(* CODESYS project silver-waffle
   Author: Robert Budgen
   Company: Burkert
   DefaultNamespace: Burkert
   LanguageModelAttribute: qualified-access-only
   Placeholder: Burkert
   Title: Burkert Device Library
   Version: 1.0.0.42

Project tree, tasks and I/O mapping:
  libraries: CAA Types Extern, 3.5.17.0 (CAA Technical Workgroup); CAA Behaviour Model, 3.5.19.0 (CAA Technical Workgroup); CAA FB Factory, 3.5.19.0 (CAA Technical Workgroup); Standard, 3.5.18.0 (System); Util, 3.5.21.0 (System); CmpBitmapPool, 3.5.17.0 (System); VisuDialogs, * (System); MemoryUtils, 3.5.18.0 (3S - Smart Software Solutions GmbH); CAA Memory, 3.5.17.0 (CAA Technical Workgroup); SysTimeRtc, 3.5.20.0 (System); CAA CiA 405, 4.1.0.0 (CAA Technical Workgroup); IoDrvEtherNetIPAdapter, 4.7.0.0 (CODESYS); IoDrvEtherNetIP, 4.7.0.0 (CODESYS); BUILDING, 1.0.0.0 (OSCAT); BASIC, 3.3.4.0 (OSCAT); FloatingPointUtils, 3.5.21.0 (System); 3S CANopenStack, 4.3.0.0 (CODESYS); IoDrvModbusTCP, 4.4.0.0 (CODESYS); Recipe Management, * (System)
  00000000-0000-0000-0000-000000000000|D:\CoDeSys\LibrariesV3\trunk\Intern\CAA\CAA Template\3.2.0.3 draft\Prefix.pdf
  00000000-0000-0000-0000-000000000000|D:\CoDeSys\LibrariesV3\trunk\Intern\CAA\CAA Template\3.4.0.0 draft\Placeholder.xml
  00000000-0000-0000-0000-000000000000|D:\CoDeSys\LibrariesV3\trunk\Intern\CAA\CAA Template\3.5.2.0 draft\Placeholder.xml
  10 Documentation/
    AL1342
    ASi_8694
    Burkert_8050
    CanOpen_8694
  20 Program Organization Units/
    function block ACV_Temp_Loop_UDFB [CFC]
    function block Basic_Temp_LOOP [CFC]
    function block BCV_Temp_Loop_UDFB [CFC]
    function block FIT_DINT_UDBF [LD]
    function block FLOWave_UDFB [CFC]: Alarms, Translate
    Helpers/
      function block CalculateFrequencyWithTime [ST]
      function block Count_to_Hz [CFC]
      function block FB_DilutionCalculator [ST]
      function block FB_LookUp_Table [ST]: GetVarY
      function block FB_TempCorrection [ST]: GetCorrection
      function Flow_ETA [ST]
      program PLC_TIME [ST]
      function RCP_Manager [ST]: LoadAndWrite, ReadAndSave
      function block Virtual_FIT [CFC]
    HMI_Sync/
      Level_0/
        CanOpen/
        eDip/
        function HMI_8228_Sync [ST]
        function block HMI_8605_Sync [ST]
        function HMI_8653_Sync [ST]
        function HMI_ME44AI_Sync [ST]
        function HMI_ME64_Sync [ST]
      Level_1/
        function block ACV_HMI_Sync_UDFB [?]
        function block AIT_HMI_Sync_UDFB [?]
        ASi/
        function block B8050_HMI_Sync_UDFB [?]
        function block BCV_HMI_Sync_UDFB [?]
        function block c8691_HMI_Sync_UDFB [?]
        function block c8694_HMI_Sync_UDFB [?]
        CanOpen/
        function block Contactor_HMI_Sync_UDFB [?]
        function block DI_HMI_Sync_UDFB [?]
        function block DO_HMI_Sync_UDFB [?]
        eDip/
        function block eDip_s8228_HMI_Sync [?]
        function block FB_HMIAlarmBinder [ST]
        function block FIT_HMI_Sync_UDFB [?]
        function block s336x_HMI_Sync [?]
        function block s8050_HMI_Sync [?]
        function block s8098_HMI_Sync_UDFB [?]
        function block s8312_HMI_Sync [?]
        function block s8412_HMI_Sync [?]
        function block SV_HMI_Sync [?]
        VFDs/
      Level_2/
        function block Chase_HMI_Sync_UDFB [?]
        function block Condensate_HMI_Sync_UDFB [?]
        function block PID_HMI_Sync_UDFB [?]
        function block Quick_Mix_HMI_Sync_UDFB [?]
        function block SW_HMI_Sync_UDFB [?]
      Level_3/
        function block Brite_HMI_Sync [?]
        function block Fermenter_HMI_Sync [?]
    Level_0_Remote_IO/
      Advantech/
        function Adam_6015_FB [LD]
        function Adam_6050_FB [LD]
        function Adam_6217_FB [LD]
        function Adam_6250 [ST]
        function Adam_6266_FB [LD]
      ASI/
        function block AC2916_AIT [LD]
      Burkert/
        function eDip_8653_UDFB [?]
        function block eDip_ME64_CTRL [ST]
        function block eDip_ReadDDO [ST]
        function block eDip_ReadDSO [ST]
        function block eDip_ReadSingleItem [ST]
        function block eDip_WriteSingleItem [ST]
        function block ME43_SDO [ST]
        function ME44_DI [ST]
      CanOpen/
        function block CanOpen_8605 [ST]
        function block CanOpen_8653 [ST]
        function block CanOpen_ME64 [ST]
        data type cSDO_DUT
      eDip/
        function block eDip_8605_CTRL [ST]
        function eDip_ME44_AI [ST]
        function eDip_ME44_AO [ST]
        function eDip_ME44_DI [ST]
        function eDip_ME44_DO_Analog [ST]
        function eDip_ME44_DO [ST]
        function block Parse_DDO [ST]
        function block Parse_DSO [ST]
      IFM/
        function block AL1340_UDFB [ST]
        function block AL1342_UDFB [ST]
      Stride/
        function block MB0_RTD [ST]
        function block SIO_MB12CDR [ST]
      Wago/
        function Wago_750_1405 [ST]
        function Wago_750_1504 [ST]
        function Wago_750_496 [ST]
        function Wago_750_555 [ST]
    Level_1_Devices/
      Asi/
        function block ACV_ASI_CTRL_UDFB [?]
        function block B8681_ASI_UDFB [CFC]
        function block BCV_ASI_CTRL_UDFB [?]
      Base_Functions/
        function block Analog_Alarm_UDFB [ST]
        function block Analog_Sensor_UDFB [?]
        function block Basic_ACV_UDFB [?]
        function block Basic_BCV_UDFB [ST]
        function block Basic_FIT [?]
        function block BCV_CTRL_UDFB [?]
        function block Contactor_Control_UDFB [CFC]
        function block DI_UDFB [CFC]
        function block DO_UDFB [CFC]
        function block LS_UDFB [ST]
      CanOpen/
      eDip/
      function block FIT_Count_UDFB [?]
      function block FIT_Rate_UDFB [?]
      function block FIT_UDFB [?]
      IoLink/
      MbTCP/
      Pumps/
      VFDs/
      Wago/
    Level_2_Controls/
      function block Analog_Batch_Pump [CFC]
      function block Analog_Control_UDFB [LD]
      function block Batch [ST]
      function block Batch_Transfer [SFC]
      function block Chase_Master_Rate_UDFB [SFC]
      function block Chase_Master_UDFB [SFC]
      function block Chase_Slave_UDFB [ST]
      function block Condensate_Trap_UDFB [CFC]
      function block DofMaster [ST]
      function block Duplex_VFD [ST]
      function block fb_ACV_Filter [ST]
      function block Filter_Pair [ST]
      function block HighSpeed_Tempered [ST]
      function block MixLine_PCT [ST]
      function block MixLine_Time [ST]
      function block PID_UDFB [CFC]
      function block Quick_Mix_UDFB [SFC]
      function block Rate_Batch [ST]
      function block SSR_Heater [ST]
      function block Stack_Lights_4Way [CFC]
      function block SW_CTRL [ST]
      function block Tempered_Line_4_Valve [ST]
      function block Tempered_Mix_UDFB [CFC]
    Level_3/
      Brewery/
    Simulators/
      function block c8691_CanOpen_Sim [ST]
      function c8694_CanOpen_Sim [ST]
      function CalculateMixedConductivity [ST]
      function CanOpen_8694_Data_Sim [ST]
      function block Contactor_Sim [ST]
      function Eaton_DM1_Sim [ST]
      function eDip_8412_Sim [ST]
      function Edip_8691_Sim [ST]
      function Edip_8694_Data_Sim [ST]
      function eDip_ME44_DI_Count_Sim [ST]
      function eDip_ME44_DI_Hz_Sim [ST]
      function FIT_Sim [ST]
      function HTX_Sim [ST]
      function Mix_Sim [ST]
      function Mix_TT_Sim [ST]
      function PipePressure [ST]
      function SSR_Heater_Sim [ST]
      function Tank_Sim [ST]
      function TankCND [ST]
      function TT_SIM [ST]
      function block Vacon_VFD_SIM [ST]
      function VFD_GS2x_Sim [ST]
      function block Volume_Sim [ST]
    function block Tempered_Mix_eDip_UDFB [CFC]
    function block Transfer_ACV_FIT_UDFB [CFC]
    function block Transfer_ACV_VFD_FIT_UDFB [CFC]
    function block Transfer_BCV_FIT_UDFB [CFC]
    function block Transfer_BCV_VFD_FIT_UDFB [CFC]
  30 Visualizations/
    image pool ImagePool
    global variables VISU
  40 Data Types/
    ASi/
      data type AC2916_DUT
      data type ASi_8694
      data type ASi_8694_PDO
      data type Asi_Node_DUT
      data type B8691_Asi_DUT
    Base_Declarations/
      global variables ASI
      data type cBase_FIT
      global variables GVL
      global variables HMI
      global variables Network
      global variables PVL
      global variables RIO
      data type Vacon_MbTCP
      data type Word_as_Real_DUT
    Brewery/
      Cellar/
      CIP/
      CLT/
      Common/
      data type Config_DUT
      Grain_Room/
      HLT/
      KT/
      LT/
      MM/
      data type Recipe_4_Vessel
      WP/
    HMI/
      Level_0/
      Level_1/
      Level_2/
      Level_3/
    Level_0_Remote_IO/
      8605/
      8653/
      Adam_6050/
      Adam_6217/
      Adam_6250/
      Asi/
      data type eDip_MEx3_ORF
      IO-Link/
      ME44_AI/
      ME44_AO/
      ME44_DI/
      ME44_DO/
      ME64/
      SIO-MB04RTDS/
      SIO-MB12CDR/
    LeveL_1_Devices/
      Base/
      data type cACV
      data type cAIT
      data type cBCV
      data type cFIT
      data type Contactor_DUT
      data type cSensor
      data type DI_DUT
      data type DO_DUT
      IO-Link/
      Networked/
      data type SV_DUT
      VFD's/
    Level_2_Functions/
      data type Analog_Control_DUT
      data type c4Way_Stack_Light
      data type cAnalog_Batch_Pump
      data type cAnalog_Batch_Pump_Config
      data type cChase
      data type cCondensate_Trap
      data type cDuplex
      data type cFilters
      Chase/
      data type cSSR
      data type cSSR_Heater
      data type cSSR_Phase
      data type cStack_Light
      Filter/
      Mix/
      data type Mix_Config_DUT
      data type Mix_DUT
      PID/
      data type Positioner_Config_DUT
      data type Positioner_DUT
      Tempered/
    Level_3/
      data type cBatch
      data type cDOF_Line_PCT
      data type cDOF_Line_Time
      data type cDOF_Master
      data type FV_DUT
    To be Sorted/
      data type ACV_eDip
      data type ACV_Temp_Loop_DUT
      data type Analog_Alarm
      data type Analog_PT_Sensor_DUT
      data type Analog_Sensor_DUT
      data type Analog_TT_Sensor_DUT
      data type Analog_Valve_DUT
      data type b336x_Config
      data type b336x_Valve_DUT
      data type B_8605_DUT
      data type BCV_Temp_Loop_Config_DUT
      data type BCV_Temp_Loop_DUT
      data type Binary_Valve_DUT
      data type c8694_PDin
      data type cAcyclic_Message
      data type cAcyclic_Request
      data type cAcyclic_Response
      data type cFLOWave_DUT
      data type CM_CR2032_PDO_DUT
      data type CM_CR2032_PDO_IN_DUT
      data type CM_CR2032_PDO_OUT_DUT
      data type cRecipe
      data type eAcyclic_Response
      data type ESL_MSG_DUT_1
      data type ESL_MSG_DUT
      data type FIT_Transfer_DUT
      data type FIT_VFD_Transfer_DUT
      data type HSC_16Bit
      data type HSC_32Bit
      data type HSC_Data_16Bit
      data type HSC_Data_32Bit
      data type HSC_DUT
      data type Lock_DUT
      data type Profile_DUT
      data type PT_Config_DUT
      data type Pump_PID_DUT
      data type Steam_Set_Config_DUT
      data type Steam_Set_DUT
      data type Tank_Lights_DUT
      data type TT_Config_DUT
      data type Valve_3285_DUT_1
      data type Valve_3285_DUT
      data type Vessel_Config_Dut
      data type Vessel_DUT
      data type Vessel_PB_DUT
  50 Functions/
    function Alarm_Offset_Convert [ST]
    function Alarm_Window_Convert [ST]
    function Anton_Parr_Deox [CFC]
    Asi/
      function block AC2916 [CFC]
      function block Asi_GW_FUN [ST]
    function ASi_8694_Mapping [CFC]
    function block b8619_CND_FB [ST]
    function block B8619_Input_FB [ST]
    function block B8619_Main_FB [ST]
    function block b8619_PH_ORP_FB [ST]
    function Build_ORF_Index [ST]
    Calculators/
      function Calc_SaltPumpSpeed [ST]
      function Calculate_Chlorine_Volume [ST]
      function DilutionOutput [ST]
      function KV_Calculator [ST]
      function MidPoint [ST]
      function VolumeBasedDilution [ST]
    function Contactor_Control_FB [CFC]
    function DaySeconds [?]
    function Find_Real_In_Array [ST]
    function FindClosestIndex [ST]
    function FindClosestIndexSorted [ST]
    function FlowWave_Mapping [LD]
    function fNord_Control_Word [LD]
    function fNord_Status_Mapping [LD]
    NVL/
      function f_Fermenter_To_NVL [ST]
    function Tempered_Flow_Calculator [ST]
    function Tempered_Look_UP [ST]
    function Unit_Convert [ST]
    function block V_Flow [CFC]
    function WORD_2_REAL_1 [LD]
    function Word_2_Real_Div [CFC]
  5ce3da45-db07-42e7-a21c-a00fff4ed8f6|C:\Users\robert.budgen.CALT0351M\Pictures\HMI Images\Tank_800h.png
  5ce3da45-db07-42e7-a21c-a00fff4ed8f6|C:\Users\robert.budgen.CALT0351M\Pictures\HMI Images\Tube Body_61x100.png
  60 Unions/
    Helpers/
      data type Bytes_2_Int
      data type bytes_2_real
      data type Bytes_DWord
      data type Bytes_Word
      data type IFM_Status
      data type ORF
      data type REAL_2_WORD
      data type uNamur
      data type uUser_Confirm
      data type WORD_2_Real
    Level_0/
    Level_1/
      data type uACV_Mode
      data type uACV_Status
      data type uAIT_Mode
      data type uAnalog_Pump_Modes
      data type uAnalog_Pump_Status
      data type uBCV_Mode
      data type uBCV_Status
      data type uContactor_Modes
      data type uDI_Mode
      data type uDI_Status
      data type uDo_Modes
      data type uDuplex_mode
      data type uHOA_Mode
      data type uM_Pump_Modes
      data type uM_Pump_Status
      data type uNord_Data_In
      data type uNord_Status_Word
      data type uSensor_Status
      data type uVFD_Mode
      data type uVFD_Status
    Level_2/
      data type uBatch_Transfer_Mode
      data type uChase_Status
      data type uHighSpeed_Tempered_Mode
      data type uHighSpeed_Tempered_Status
      data type uHighSpeed_Tempered_Task
      data type uPID_Modes
      data type uPID_Status
      data type uQuick_Mix_Modes
      data type uTempered_Modes
      data type uTempered_Status
      data type uTempered_Tasks
    Level_3/
      data type uBatch_Status
      data type uBatch_Task
      data type uBrite_Modes
      data type uBrite_Status
      data type uCLT_Mode
      data type uCLT_Status
      data type uCLT_Task
      data type uFermenter_Modes
      data type uFermenter_Status
      data type uFilter_Manager_Modes
      data type uFilter_Status
      data type uFilterMode
      data type uGR_Status
      data type uGR_Task
      data type uHLT_Mode
      data type uHLT_Status
      data type uHLT_Task
      data type uKT_Mode
      data type uKT_Status
      data type uKT_Task
      data type uLT_Mode
      data type uLT_Task
      data type uMM_Mode
      data type uMM_Task
      data type uWP_Mode
      data type uWP_Modes
      data type uWP_Status
      data type uWP_Task
    data type uService_Water_Destination
  70 Modes Enums/
    Brewery/
      data type BH_Vessel_Modes
      data type CIP_1_Modes
      data type eBrite_Modes
      data type eCLT_Modes
      data type eFermenter_Modes
      data type eGR_Modes
      data type eHLT_Modes
      data type eKT_Mode
      data type eLT_Modes
      data type eMM_Modes
      data type FV_Modes
      data type HLT_Blending_Modes
      data type KTWP_Modes
      data type MM_Decoction_Modes
    Level_0/
      data type eMB0_RTD_Input_Type
      data type eMB0_RTD_Units
      data type Reset_Relay_Mode
    Level_1/
      data type AIT_Modes
      data type Command_Modes
      data type Contactor_Modes
      data type Di_Modes
      data type DO_Modes
      data type e_8681_Modes
      data type eACV_Modes
      data type eAnalog_Control_Modes
      data type eAnalog_Pump_Modes
      data type eAODD_Modes
      data type eB336x_Modes
      data type eBCV_Modes
      data type eConfig_startTune
      data type eHOA_Modes
      data type eM_Pump_Modes
      data type Fan_Modes
      data type LS_Modes
      data type Positioner_Modes
      data type PT_Modes
      data type TT_Modes
      data type VFD_Modes
    Level_2/
      data type AIT_Transfer_Modes
      data type eBatch_Transfer_Mode
      data type eChase_Mode
      data type eDuplex_Mode
      data type eFilter_Manager_Modes
      data type eFilter_Mode
      data type eHighSpeed_Tempered_Mode
      data type ePID_Modes
      data type eQuick_Mix_Modes
      data type eTempered_Modes
      data type FIT_Transfer_Modes
      data type FIT_VFD_Transfer_Modes
      data type Mix_Modes
      data type Steam_Condensate_Modes
      data type Steam_Modes
      data type Temp_loop_Modes
    Level_3/
      data type CLT_Modes
      data type eKT_Modes
      data type eRCP_Mode
      data type eWP_Modes
  80 Status Enums/
    Level_0/
      data type eNamur107
      data type eORF_Status
      data type SDO_Error_Codes
    Level_1/
      data type Contactor_Status
      data type DI_Status
      data type DO_Status
      data type e8691_ValveMode
      data type e8691_xTuneStatus
      data type e8694_xTuneStatus
      data type eACV_Status
      data type eAnalog_Pump_Status
      data type eAODD_Status
      data type eB8681_Status
      data type eBCV_Status
      data type eCurrentOpMode
      data type eFloWave_Status
      data type eM_Pump_Status
      data type eSensor_Status
      data type eVFD_Status
      data type Positioner_Status
      data type PT_Status
      data type SV_Status
      data type TT_Status
      data type VFD_Fault_Status
    Level_2/
      data type eChase_Status
      data type eCondensate_Status
      data type eFilter_Manager_Status
      data type eFilter_Status
      data type eHighSpeed_Tempered_Status
      data type ePID_Status
      data type eQuick_Mix_Status
      data type eTempered_Status
      data type Mix_Status
      data type Temp_loop_Status
      data type Transfer_Status
    Level_3/
      data type eBatch_Status
    Vessels/
      data type BH_Vessel_Status
      data type eBrite_Status
      data type eCLT_Status
      data type eFermenter_Status
      data type eGrain_Room_Status
      data type eHLT_Status
      data type eKT_Status
      data type eLT_Status
      data type eMM_Status
      data type eWP_Status
  90 Task Enums/
    data type eCLT_Task
    data type eFilter_Task
    data type eGR_Task
    data type eHighSpeed_Tempered_Task
    data type eHLT_Task
    data type eKT_Task
    data type eLT_Task
    data type eMEx3SDO
    data type eMM_Task
    data type eTempered_Task
    data type eWP_Task
    Level_3/
      data type eBatch_Task
  eNum_notifications/
    data type eHLT_Notifications
    data type eMM_Notifications
    data type eUnits
    data type eUser_Confirm
  text list GlobalTextList
  Library Information/
    function GetLibVersion [ST]
    function GetLibVersionNumber [ST]
    function IsLibReleased [ST]
  function GetBooleanProperty [ST]
  function GetCompany [ST]
  function GetTextProperty2 [ST]
  function GetTextProperty [ST]
  function GetTitle [ST]
  function GetVersion [ST]
  function GetVersionProperty [ST]
*)

// 60 Unions/uService_Water_Destination
TYPE uService_Water_Destination :
UNION
	iTarget:INT;
	eTarget:Service_Water_Mapping;
END_UNION
END_TYPE

// 90 Task Enums/eCLT_Task
{attribute 'qualified_only'}
//{attribute 'strict'}
{attribute 'to_string'}
TYPE eCLT_Task :
(
	Off :=0,						
	Fill, 													
	Cool_Recirculate,
	Ready_Holding,
	Ready,		
	Line_Chase,				
		
	Spray_Ball,
	Fill_Cool
		

	
);
END_TYPE

// 90 Task Enums/eFilter_Task
{attribute 'qualified_only'}
{attribute 'strict'}
TYPE eFilter_Task :
(
	Off := 0,
	Standby,
	Drain,
	Flush,
	InService,
	Bypass
	
);
END_TYPE

// 90 Task Enums/eGR_Task
{attribute 'qualified_only'}
//{attribute 'strict'}
{attribute 'to_string'}
TYPE eGR_Task :
(
	OFF := 0,
	Dispense
);
END_TYPE

// 90 Task Enums/eHighSpeed_Tempered_Task
{attribute 'qualified_only'}
{attribute 'strict'}
TYPE eHighSpeed_Tempered_Task :
(
	OFF := 0,
	Calibrate,
	Run
);
END_TYPE

// 90 Task Enums/eHLT_Task
{attribute 'qualified_only'}
//{attribute 'strict'}
{attribute 'to_string'}
TYPE eHLT_Task :
(
	Off :=0,						
	Fill, 													
	Heat_Recirculate,
	Ready_Holding,
	Ready,		
	Line_Chase,				
		
	Spray_Ball,
	Fill_Heat			

	
);
END_TYPE

// 90 Task Enums/eKT_Task
{attribute 'qualified_only'}
//{attribute 'strict'}
{attribute 'to_string'}
TYPE eKT_Task :
(
	OFF := 0,
	PreHeat,
	Wort_In,
	Full_Boil,
	Jacket_Boil,
	Rocket_Boil,
	Transfer,
	Transfer_Chase,
	Quick_Rinse, //8
	Tank_Drain,
	Transfer_in,
	Whirlpool,
	Rest,
	Transfer_Out,
	Turb_Buster, //14
	Drain,		//15
	Mash_In_Rocket_Transition,
	Mash_In_Rocket
);
END_TYPE

// 90 Task Enums/eLT_Task
{attribute 'qualified_only'}
//{attribute 'strict'}
{attribute 'to_string'}
TYPE eLT_Task :
(
	Off :=0,
	Move_Brew_Configuration,	//
	Foundation_Water,
	Mash_In,
	
	First_Underlet,	//4
	Second_Underlet,
	Third_Underlet,
	
	First_Vorlauf,	//7
	Second_Vorlauf,
	Third_Vorlauf,
	
	First_Transfer,	//10
	Second_Transfer,
	Third_Transfer,
	
	First_Sparge,	//13
	Second_Sparge,
	Third_Sparge,
	
	Transfer_Empty,	//16
	Transfer_Chase,		//17
	Tank_Clean,
	Quick_Rinse,		//19
	Tank_Drain,			//20
	Spent_Grain,		//21
	CIP,
	Pre_Heat			//23
	
					
	
	
);
END_TYPE

// 90 Task Enums/eMEx3SDO
{attribute 'qualified_only'}
{attribute 'strict'}
TYPE eMEx3SDO :
(
	Idle := 0,
	GW_Read_Configure,
	GW_Read,
	GW_Evaluate,
	Node_Read_Configure,
	Node_Read,
	Node_Evaluate,
	
	
	Scan,
	Scan_Configure,
	Scan_Read,
	Scan_Evaluate,
	Scan_Clear,
	
	
	NamurNe107,
	Temperature,
	Voltage,
	Operation_Time,
	Ident,
	Product_Code,
	Serial_Number,
	
	
	TravelACC,
	ValveCycles,
	TuneStarts,
	PilotCycles,
	
	
	End_task
	
);
END_TYPE

// 90 Task Enums/eMM_Task
{attribute 'qualified_only'}
//{attribute 'strict'}
{attribute 'to_string'}
TYPE eMM_Task :
(
	Off :=0,					
	Confirm,
	//Confirmed,
	Preheat,
	Mash_In,	//3						
	Heat_1,		//4
	Heat_2,
	Heat_3,
	//Heat_4,
	//Mash_Complete,				
	Mash_Out,		//7			
	//Transfer_Complete,			
	Transfer_Flush,		//8		
	//Transfer_Flush_Complete,	
	Quick_Rinse,	//9			
	//Quick_Rinse_Complete,		
	Drain,			//10			
	//Drain_Complete,				
	
	//CIP_Fill,					
	//CIP_Fill_Complete,			
	//CIP_Recirculate,			
	//CIP_Recirculate_Complete,	
	//CIP_Transfer,				
	//CIP_Transfer_Complete,		
	//CIP_Transfer_Flush,			
	//CIP_Transfer_Flush_Complete 
	CIP,
	Vorlauf,
	Transfer,
	Transfer_Sparge,
	Fly_Sparge,
	UnderLet,
	Foundation,	//17
	Grain_Out
	

	
	
);
END_TYPE

// 90 Task Enums/eTempered_Task
{attribute 'qualified_only'}
//{attribute 'strict'}
{attribute 'to_string'}
TYPE eTempered_Task :
(
	OFF := 0,
	Calibrate,
	Run,
	Drain,
	Prime
	//Rinse
	
);
END_TYPE

// 90 Task Enums/eWP_Task
{attribute 'qualified_only'}
{attribute 'to_string'}
TYPE eWP_Task :
(
	Off :=0, 						//0
	Transfer_in,
	Whirlpool,
	Rest,
	CastOut,
	CastOut_Chase,
	Trub_Buster,
	Quick_Rinse,
	Tank_Drain
	
);
END_TYPE

// eNum_notifications/eHLT_Notifications
{attribute 'qualified_only'}
{attribute 'strict'}
TYPE eHLT_Notifications :
(
	System_OK,
	Pump_Not_In_Auto,
	Pump_Faulted,
	HTX_Valve_Not_In_Auto,
	Recirc_Valve_Not_In_Auto,
	Spray_Ball_Valve_Not_In_Auto,
	Refill_Valve_Not_In_Auto,
	Pump_Intake_Empty
	
);
END_TYPE

// eNum_notifications/eMM_Notifications
{attribute 'qualified_only'}
{attribute 'strict'}
TYPE eMM_Notifications :
(
	System_OK := 0,
	Pump_Fault,
	Pump_Not_In_Auto
);
END_TYPE

// eNum_notifications/eUnits
{attribute 'qualified_only'}
{attribute 'to_string'}
TYPE eUnits :
(
	None := 0,
	bar,
	psi,
	in_H20,
	pa,
	
	C,
	F,
	K,
	
	l,
	USg,
	m3,
	
	lps,
	lpm,
	gpm,
	m3_min,
	
	S_CM,
	S_M,
	uS_cm,
	mS_cm,
	ppm,
	
	
	Kohm_cm,
	mg_l,
	
	
	
	
	
	
	Raw
);
END_TYPE

// eNum_notifications/eUser_Confirm
{attribute 'qualified_only'}
//{attribute 'strict'}
TYPE eUser_Confirm :
(
	Hidden := 0,
	Confirm,
	Confirmed
);
END_TYPE

// 40 Data Types/ASi/AC2916_DUT
TYPE AC2916_DUT :
STRUCT
	Detected:BOOL;
	PROJECTED:BOOL;
	Active:BOOL;
	Fault:BOOL;
	AI:ARRAY[1..4] OF WORD;
END_STRUCT
END_TYPE

// 40 Data Types/ASi/ASi_8694
TYPE ASi_8694 EXTENDS cACV :
STRUCT
	PDO:ASi_8694_PDO;
END_STRUCT
END_TYPE

// 40 Data Types/ASi/ASi_8694_PDO
TYPE ASi_8694_PDO :
STRUCT
	Actual:REAL;
	Output:REAL;
END_STRUCT
END_TYPE

// 40 Data Types/ASi/Asi_Node_DUT
TYPE Asi_Node_DUT :
STRUCT
	Detected:BOOL;
	PROJECTED:BOOL;
	Active:BOOL;
	Fault:BOOL;
	Analog_RX_0:WORD;
	Analog_RX_1:WORD;
	Analog_TX_0:WORD;
	Analog_TX_1:WORD;
	Digital_RX:BYTE;
	Digital_TX:BYTE;
	
	
END_STRUCT
END_TYPE

// 40 Data Types/ASi/B8691_Asi_DUT
TYPE B8691_Asi_DUT :
STRUCT
	Mode	:	e_8681_Modes;
	Status	:	WORD;
	HMI_CMD	:	INT;
	PLC_CMD	:	INT;
	Status1 :eB8681_Status;
	Valve_Status:BYTE;
END_STRUCT
END_TYPE

// 40 Data Types/Base_Declarations/cBase_FIT
TYPE cBase_FIT :
STRUCT
	Rate:cSensor;
	Total:REAL;
	PLC_Reset:BOOL;
	//Counts	:	UDINT;
	//Frequency	:REAL;
	K:REAL;
	HMI_Reset:BOOL;
END_STRUCT
END_TYPE

// 40 Data Types/Base_Declarations/Vacon_MbTCP
TYPE Vacon_MbTCP :
STRUCT
	RX : ARRAY[0..10] OF WORD; 
	TX : ARRAY[0..2] OF WORD; 
END_STRUCT
END_TYPE

// 40 Data Types/Base_Declarations/Word_as_Real_DUT
TYPE Word_as_Real_DUT :
UNION
	Words:ARRAY[0..1] OF WORD;
	rReal:REAL;
END_UNION
END_TYPE

// 40 Data Types/Brewery/Config_DUT
TYPE Config_DUT :
STRUCT
	HLT:HLT_DUT;
	CLT:CLT_DUT;
	Grain_Room:GR_DUT;
	MM:MM_DUT;
	LTun:LT_DUT;
	KT:cKT;
	WP:cWP_DUT;
	Brew_Recipe:INT;
END_STRUCT
END_TYPE

// 40 Data Types/Brewery/Recipe_4_Vessel
TYPE Recipe_4_Vessel :
STRUCT
	MM:cMM_Recipe;
	LTun:cLT_Recipe;
	KT:cKT_Recipe;
	WP:cwp_recipe;
	
END_STRUCT
END_TYPE

// 40 Data Types/Level_0_Remote_IO/eDip_MEx3_ORF
TYPE eDip_MEx3_ORF :
STRUCT
	Call:WORD;
	Index_TX:DWORD;
	Index_RX:DWORD;
	Result:DWORD;
	Length:DWORD;
	Value_TX:DWORD;
	Value_RX:DWORD;
	Write_Value:BOOL;
	Device_Status:UINT;
	Control_Word:Bytes_Dword;
	CommState:ModbusTCPComState;
	Restart:BOOL;
	
	strTCPstate:STRING[30];
END_STRUCT
END_TYPE

// 40 Data Types/LeveL_1_Devices/cACV
TYPE cACV :
STRUCT
	HMI_CMD:REAL;
	PLC_CMD:REAL;
	Valve_Actual:REAL;

	Mode:uACV_Mode;//ACV_Modes;
	Status:uACV_Status;
	Ready:BOOL;

END_STRUCT
END_TYPE

// 40 Data Types/LeveL_1_Devices/cAIT
TYPE cAIT:// EXTENDS cSensor :
STRUCT
	Sensor			:	cSensor;
	Analog_Scale	:	cAnalog_scale;
	
END_STRUCT
END_TYPE

// 40 Data Types/LeveL_1_Devices/cBCV
TYPE cBCV :
STRUCT
	Mode	:uBCV_MODE;
	PLC_CMD	:	BOOL;
	Status:	uBCV_Status;
	Ready:BOOL;

		
END_STRUCT
END_TYPE

// 40 Data Types/LeveL_1_Devices/cFIT
TYPE cFIT EXTENDS cBase_FIT :
STRUCT

	Counts	:	UDINT;
	Frequency	:REAL;

END_STRUCT
END_TYPE

// 40 Data Types/LeveL_1_Devices/Contactor_DUT
TYPE Contactor_DUT :
STRUCT
	Mode:uContactor_Modes;
	Status:Contactor_Status;
	PLC_CMD_FWD:BOOL;
	PLC_CMD_Rev:BOOL;
	Q1:BOOL;
	Q2:BOOL;
	
END_STRUCT
END_TYPE

// 40 Data Types/LeveL_1_Devices/cSensor
TYPE cSensor :
STRUCT
	Alarm_Config	:	cAlarm_Config;
	
	EU:		REAL;
	Ready:	BOOL;
	
	Status:uSensor_Status;
	
	Mode			:	uAIT_Mode;
	Force_Value:REAL;
	
END_STRUCT
END_TYPE

// 40 Data Types/LeveL_1_Devices/DI_DUT
TYPE DI_DUT :
STRUCT
	MODE:uDi_Mode;
	Status:uDi_Status;
	Raw:BOOL;
	Q:BOOL;
END_STRUCT
END_TYPE

// 40 Data Types/LeveL_1_Devices/DO_DUT
TYPE DO_DUT :
STRUCT
	Mode:uDO_Modes;
	Status:DO_Status;
	Q:BOOL;
	PLC_CMD:BOOL;
	Ready:BOOL;
END_STRUCT
END_TYPE

// 40 Data Types/LeveL_1_Devices/SV_DUT
TYPE SV_DUT :
STRUCT
	Mode:uBCV_Mode;
	Status:uBCV_Status;
	Q:BOOL;
	PLC_CMD:BOOL;
	Ready:BOOL;
	Namur:uNamur;
	strNamur:STRING[30];
END_STRUCT
END_TYPE

// 40 Data Types/Level_2_Functions/Analog_Control_DUT
TYPE Analog_Control_DUT :
STRUCT
	Alarm_Config	:	cAlarm_Config;
	Analog_Scale	:	cAnalog_scale;
	Mode			:	eAnalog_Control_Modes;
	EU:		REAL;
	PLC_Target:REAL;
	HMI_Target:REAL;
	output:REAL;
	Status:eSensor_Status;
END_STRUCT
END_TYPE

// 40 Data Types/Level_2_Functions/c4Way_Stack_Light
TYPE c4Way_Stack_Light :
STRUCT
	RED:cStack_light;
	Yellow:cStack_Light;
	Green:cStack_Light;
	Horn:cStack_light;
END_STRUCT
END_TYPE

// 40 Data Types/Level_2_Functions/cAnalog_Batch_Pump
TYPE cAnalog_Batch_Pump EXTENDS cAnalog_Pump : 
STRUCT
	//Mode:eAnalog_Pump_Modes;
	Config:cAnalog_Batch_Pump_Config;
	HMI_Volume_Target:REAL;
	PLC_Volume_Target:REAL;
	
	Live_Rate:REAL;
	Volume_Delivered:REAL;
	PCT_Remain:REAL;
	Batch_ETA:INT;
	
END_STRUCT
END_TYPE

// 40 Data Types/Level_2_Functions/cAnalog_Batch_Pump_Config
TYPE cAnalog_Batch_Pump_Config :
STRUCT
	//Base_Rate_LPM:REAL:=10;
	Min_Speed:REAL:=15;
	Max_Speed:REAL:=100;
	SuckBack_Speed:REAL:=10;
	SuckBack_Seconds:INT:=3;
	Available_Volume:REAL:=0;
	Follow_Rate:REAL;
	Follow_ENABLE:BOOL;
END_STRUCT
END_TYPE

// 40 Data Types/Level_2_Functions/cChase
TYPE cChase :
STRUCT
	Target_Rate:REAL;
	Target_Volume:REAL;
	Target_Temp:REAL;
	PCT_Remain:REAL;
	ETA:UINT;
	Mode:INT;
	PLC_Run:BOOL;
	Active:BOOL;
	Status:uChase_Status;
END_STRUCT
END_TYPE

// 40 Data Types/Level_2_Functions/cCondensate_Trap
TYPE cCondensate_Trap :
STRUCT
	LSHH:DI_DUT;
	LSH:DI_DUT;
	LSL:DI_DUT;
	LSLL:DI_DUT;
	Min_Valve_Positions:ARRAY[0..3] OF REAL;
	CV:REAL;
	READY:BOOL;
	Status:eCondensate_Status;
END_STRUCT
END_TYPE

// 40 Data Types/Level_2_Functions/cDuplex
TYPE cDuplex :
STRUCT
	Mode:uDuplex_mode;
	Run_Request:BOOL;
	Run_Pct:REAL;
	Target_Split:REAL;
	Current_Split:REAL;
	RunTime_1:TIME;
	RunTime_2:TIME;
	
	
END_STRUCT
END_TYPE

// 40 Data Types/Level_2_Functions/cFilters
TYPE cFilters :
STRUCT
	Group_Mode:uHOA_Mode;
	A_Mode:uHOA_Mode;
	A_Status:eFilter_Status;
	A_Task:eFilter_Task;
	
	B_Mode:uHOA_Mode;
	B_Status:eFilter_Status;
	B_Task:eFilter_Task;
	
	DP_Alarm:cAlarm_Config;
	DP:REAL;
	
	
END_STRUCT
END_TYPE

// 40 Data Types/Level_2_Functions/cSSR
TYPE cSSR :
STRUCT
	U:cSSR_Phase;
	V:cSSR_Phase;
	W:cSSR_Phase;
	Seconds:UDINT;
	Cycles:UDINT;
	Active_Phases:BYTE;
	
END_STRUCT
END_TYPE

// 40 Data Types/Level_2_Functions/cSSR_Heater
TYPE cSSR_Heater :
STRUCT
	SSR:ARRAY[0..2] OF cSSR;
	Main_Contactor:BOOL;
	
	Min_On_Time_S:UINT;
	Min_Rest_S:UINT;
	Effective_Output:REAL;
	
	
	
	
	
	
END_STRUCT
END_TYPE

// 40 Data Types/Level_2_Functions/cSSR_Phase
TYPE cSSR_Phase :
STRUCT
	Q:BOOL;
	Request:BOOL;
	Seconds:UDINT;
	Cycles:UDINT;
END_STRUCT
END_TYPE

// 40 Data Types/Level_2_Functions/cStack_Light
TYPE cStack_Light :
STRUCT
	ON:BOOL;
	Flash_Rate_ms:UINT;
	Q:BOOL;
END_STRUCT
END_TYPE

// 40 Data Types/Level_2_Functions/Mix_Config_DUT
TYPE Mix_Config_DUT :
STRUCT
	Min_Flow:REAL;
	Max_Flow:REAL;
	Foundation_Volume:REAL;
	Foundation_Rate:REAL;
	Ramp_Rate:REAL;
	Flow_KP:REAL;
	Flow_TN:REAL;
	Flow_TV:REAL;
	
	
	Temp_KP:REAL;
	Temp_TN:REAL;
	Temp_TV:REAL;


   REMAIN_L : REAL ;
   START_lpm : REAL := 5.0 ;

   TARGET_C : REAL ;
   TARGET_L : REAL ;
   TARGET_lpm : REAL := 10.0 ;
   TEMP_WINDOW : REAL := 2.0 ;
   
	Main_ETA_S:INT;
   //	MODE : Mix_modes ;
	//Stage:UINT;
  	START_TIME_S : UINT := UINT#30 ;
   	STATUS : Mix_Status ;
   
	
	
END_STRUCT
END_TYPE

// 40 Data Types/Level_2_Functions/Mix_DUT
TYPE Mix_DUT :
STRUCT //Mainly Read Only Data for HMI
	Mode:Mix_Modes; // Read Only HMI
	Status:Mix_Status; // Read Only HMI
	Actual_Rate_EU:REAL; // Actual Rate
	Actual_Volume_EU:REAL; // Volume Dispensed
	Actual_Temp_EU:REAL;
	Flow_CV:REAL;
	Temp_CV:REAL;
	HW_CMD:REAL;
	CW_CMD:REAL;

	Grain_ETA_S:INT;
	Config:Mix_Config_DUT;
	
END_STRUCT
END_TYPE

// 40 Data Types/Level_2_Functions/Positioner_Config_DUT
TYPE Positioner_Config_DUT :
STRUCT
	Contactor:INT;
	VFD:INT;
	Pos_Min:UINT;
	Pos_Max:UINT;
	RAW:REAL;
	
END_STRUCT
END_TYPE

// 40 Data Types/Level_2_Functions/Positioner_DUT
TYPE Positioner_DUT :
STRUCT
	Mode:INT;
	Status:INT;
	Manual_Target:REAL;
	PLC_Target:REAL;
	Actual_Position:REAL;
	Closed_Limit:BOOL;
	Open_Limit:Bool;
END_STRUCT
END_TYPE

// 40 Data Types/Level_3/cBatch
TYPE cBatch :
STRUCT
	Min_Rate:REAL;
	Max_Rate:REAL;
	Start_Volume:REAL;
	End_Volume:REAL;
	
	Batch_Volume:REAL;
	Batch_Rate:REAL;
	
	Live_Target_Volume:REAL;
	Live_Target_Rate:REAL;
	
	Actual_Volume:REAL;
	Actual_Rate:REAL;
	
	
	PCT_Complete:REAL;
	System_Load:REAL;
	ETA:UINT;
	
	Ready:BOOL;
	Active:BOOL;
	
	Line_Mode:uHOA_Mode;
	Line_Task:uBatch_Task;
	Line_Status:uBatch_Status;
	PLC_Run:BOOL;
	
	StrLine_Mode:STRING;
	StrLine_Task:STRING;
	StrLine_Status:STRING;
	
	
END_STRUCT
END_TYPE

// 40 Data Types/Level_3/cDOF_Line_PCT
TYPE cDOF_Line_PCT EXTENDS cBatch :
STRUCT
	Target_PCT:REAL;
	Start_Point:REAL:=0;
	Live_PCT:REAL;
	Rate_KP:REAL:=0.1;
	
	
	
END_STRUCT
END_TYPE

// 40 Data Types/Level_3/cDOF_Line_Time
TYPE cDOF_Line_Time EXTENDS cBatch :
STRUCT
	Target_PCT:REAL;
	Live_PCT:REAL;
	Start_Time_S:UINT;
	End_Time_S:UINT;
	
	Rate_KP:REAL;
	
	
	
END_STRUCT
END_TYPE

// 40 Data Types/Level_3/cDOF_Master
TYPE cDOF_Master :
STRUCT
	
	Batch_Volume:REAL;
	Batch_Rate:REAL;
	Batch_Mode:uHOA_Mode;
	Batch_Task:uBatch_Task;
	Batch_Status:uBatch_Status;
	
	PLC_Run:BOOL;
	
	Current_Load_High:REAL;
	Current_Load_Low:REAL;
	Current_Batch_PCT:REAL;
	Batch_CLK:TIME;
	Batch_Remain:TIME;
	Current_Batch_Volume:REAL;
	Current_Batch_Rate:REAL;
	Batch_Target_ms:UDINT;
	Batch_Elapsed_ms:UDINT;
	Batch_Remain_ms:UDINT;
	Batch_ETA_ms:UDINT;
	
	
	StrBatch_Mode:STRING;
	StrBatch_Task:STRING;
	StrBatch_Status:STRING;
	
	MasterID:UDINT:=0;
	Active:BOOL;
	
	
	
	
	
END_STRUCT
END_TYPE

// 40 Data Types/Level_3/FV_DUT
TYPE FV_DUT :
STRUCT
	Mode:INT;

	Ferment_Setpoint:REAL;
	Dry_Hop_Setpoint:REAL;
	Crash_Setpoint:REAL;
	
		
		
END_STRUCT
END_TYPE

// 40 Data Types/To be Sorted/ACV_eDip
TYPE ACV_eDip :
STRUCT
	DirChanges:REAL;
	TravelAccu:REAL;
	XTunes:UINT;
	DeviceSupplyVoltage:REAL;
	DeviceTemperature:REAL;
	IdentNumber:UDINT;
	currOPmode:BYTE;
	ProductCode:UDINT;
	SerialNumber:UDINT;
	DEVmax:REAL;
	POSmonitor_Error:BYTE;
	currTUNEstatus:BYTE;
	Valve_Status:BYTE;
	
	
	
END_STRUCT
END_TYPE

// 40 Data Types/To be Sorted/ACV_Temp_Loop_DUT
TYPE ACV_Temp_Loop_DUT :
STRUCT
	Target_EU:REAL;
	DeadBand:REAL;
	Window:REAL;
	Mode:Temp_Loop_Modes;
	Timer_Target_m:UINT;
	Timer_Remaining_s:UINT;
	kp:REAL;
	TN:REAL;
	TV:REAL;
	Actual_EU:REAL;
	Error_EU:REAL;
	Live_Target_EU:REAL;
	Load_EU:REAL;
	Status:Temp_loop_Status;
	Int_Out:REAL;
	Diff_Out:REAL;
	Limiter:BOOL;
END_STRUCT
END_TYPE

// 40 Data Types/To be Sorted/Analog_Alarm
TYPE Analog_Alarm :
STRUCT
	Status	:	INT;
	//Hi_Hi_Alarm	:	BOOL;
	//Hi_Warning	:	BOOL;
	//Low_Warning	:	BOOL;
	///Low_Low_Alarm	:	BOOL;
	
	
END_STRUCT
END_TYPE

// 40 Data Types/To be Sorted/Analog_PT_Sensor_DUT
TYPE Analog_PT_Sensor_DUT :
STRUCT
	EU:		REAL;
	//Status	:	INT;
	Status:PT_Status;

END_STRUCT
END_TYPE

// 40 Data Types/To be Sorted/Analog_Sensor_DUT
TYPE Analog_Sensor_DUT :
STRUCT
	EU:		REAL;
	//Status	:	INT;
	Status:eSensor_Status;

END_STRUCT
END_TYPE

// 40 Data Types/To be Sorted/Analog_TT_Sensor_DUT
TYPE Analog_TT_Sensor_DUT :
STRUCT
	EU:		REAL;
	Status:TT_Status;

END_STRUCT
END_TYPE

// 40 Data Types/To be Sorted/Analog_Valve_DUT
TYPE Analog_Valve_DUT :
STRUCT
	Mode	: INT;
	PLC_CMD	:	REAL;
	HMI_CMD :	REAL;
	Actual	:REAL;
	Status:	UINT;
END_STRUCT
END_TYPE

// 40 Data Types/To be Sorted/b336x_Config
TYPE b336x_Config :
STRUCT
	DBDx:REAL;
	XCOdynamic:WORD;
	CHARACTselect:WORD;
	CUTOFFmin:REAL;
	CUTOFFmax:REAL;
	POSmin:REAL;
	POSmax:REAL;
	XTIMEopen:REAL;
	XTIMEclose:REAL;
	SafeposFunc:WORD;
	SafePos:REAL;
	XTUNE_error:WORD;
	XTUNE_mode:WORD;
	startTune:eConfig_startTune;
	currOPmode:WORD;
	FuncActiv:UDINT;
	ChargeFirst:WORD;
	EnergyStorageState:WORD;
END_STRUCT
END_TYPE

// 40 Data Types/To be Sorted/b336x_Valve_DUT
TYPE b336x_Valve_DUT :
STRUCT
	Mode:eB336x_Modes;
	Status:eACV_Status;
	HMI_CMD:REAL;
	PLC_CMD:REAL;
	
	Pos:REAL;
	PV:REAL;
	Valve_Status:BYTE;
	CMD:REAL;
	Setpoint:REAL;
	ExtError:BYTE;
	isPCOextern:BYTE;
	Config:b336x_Config;
	
END_STRUCT
END_TYPE

// 40 Data Types/To be Sorted/B_8605_DUT
TYPE B_8605_DUT :
STRUCT
	ActualFlow:REAL;
	AI1:REAL;
	CoilCurrent:REAL;
	DI1:BOOL;
	DI2:BOOL;
	NamurStatus:BYTE;
	Bin:BYTE;
	Fin:REAL;
	out:BYTE;
	
END_STRUCT
END_TYPE

// 40 Data Types/To be Sorted/BCV_Temp_Loop_Config_DUT
TYPE BCV_Temp_Loop_Config_DUT :
STRUCT
	Max_Cycle_S:REAL:=600;
	Min_Cycle_S:REAL:=60;
	Target_EU:REAL;
	DeadBand:REAL:=0.2;
	Window:REAL:=1;
	Mode:Temp_Loop_Modes;
	Timer_Target_m:UINT;
	Timer_Remaining_s:UINT;
	kp:REAL:=1;
	TN:REAL:=60;
	TV:REAL:=0;
	cycles:UDINT;

END_STRUCT
END_TYPE

// 40 Data Types/To be Sorted/BCV_Temp_Loop_DUT
TYPE BCV_Temp_Loop_DUT :
STRUCT
	Actual_EU:REAL;
	Error_EU:REAL;
	LIVE_Target_EU:REAL;
	Load_EU:REAL;
	Status:Temp_loop_Status;
	Max_Cycle_S:REAL:=600;
	Min_Cycle_S:REAL:=60;
	Target_EU:REAL;
	DeadBand:REAL:=0.2;
	Window:REAL:=1;
	Mode:Temp_Loop_Modes;
	Timer_Target_m:UINT;
	Timer_Remaining_s:UINT;
	kp:REAL:=1;
	TN:REAL:=60;
	TV:REAL:=0;
	cycles:UDINT;
	Output:BOOL;
	Temp_Profile:Profile_DUT;
	Int_Out:REAL;
	Diff_Out:REAL;
	Limiter:BOOL;

END_STRUCT
END_TYPE

// 40 Data Types/To be Sorted/Binary_Valve_DUT
TYPE Binary_Valve_DUT :
STRUCT
	Mode	: INT;
	PLC_CMD	:	BOOL;
	Status:	UINT;
	StrMode:eBCV_Modes;
	StrStatus:eBCV_Status;
		
END_STRUCT
END_TYPE

// 40 Data Types/To be Sorted/c8694_PDin
TYPE cDigital_ACV_PDin :
STRUCT
	Valve_Position:REAL;
	Target_Position:REAL;
	Namur_Status:e8691_Namur_Status;
	Valve_Status:e8691_Valve_Status;
	Open_Limit:BOOL;
	Close_Limit:BOOL;
	
END_STRUCT
END_TYPE

// 40 Data Types/To be Sorted/cAcyclic_Message
TYPE cAcyclic_Message :
STRUCT
	Done:BOOL;
	Request:cAcyclic_Request;
	Response:cAcyclic_Response;
END_STRUCT
END_TYPE

// 40 Data Types/To be Sorted/cAcyclic_Request
TYPE cAcyclic_Request :
STRUCT
	Port:WORD;
	Index:WORD;
	SubIndex:WORD;
	User_ID:BYTE;
	Command:BYTE;
	Length:WORD;
	Data:ARRAY[0..31] OF BYTE;
	
	
END_STRUCT
END_TYPE

// 40 Data Types/To be Sorted/cAcyclic_Response
TYPE cAcyclic_Response :
STRUCT
	Port:WORD;
	Index:WORD;
	SubIndex:WORD;
	User_ID:BYTE;
	Command:BYTE;
	Response:eAcyclic_Response;
	Length:WORD;
	Data:ARRAY[0..31] OF BYTE;
END_STRUCT
END_TYPE

// 40 Data Types/To be Sorted/cFLOWave_DUT
TYPE cFLOWave_DUT :
STRUCT
	


	Acoustic_Trans:REAL;
	AcousticImpedance:REAL;
	Concentration_1:REAL;
	Concentration_2:REAL;
	Density:REAL;
	Density_Factor:REAL;;
	Dynamic_Viscosity:REAL;
	FoulingFactor:REAL;
	Gas_Bubble_Factor:REAL;
	Kinematic_vicosity:REAL;
	Liquid_Velocity:REAL;
	Mass_Flow:REAL;
	Mass_Total_1:REAL;
	Mass_Total_2:REAL;	
	Namur_Status:INT;
	Saw_Group_Velocity:REAL;
	SpeedOfSound:REAL;
	Temp:REAL;
	Total_1:REAL;
	Total_2:REAL;
	Turbulance_Factor:REAL;
	Viscosity_Factor:REAL;
	Volume_Flow:REAL;	
	FIT_1:cFIT;
	FIT_2:cFIT;
	Status:eFloWave_Status;
	M_Reset_1:BOOL;
	M_Reset_2:BOOL;
	Alarm_Config:ARRAY[0..3] OF cAlarm_Config;
	Locate:BOOL;
	Maintenance:BOOL;
END_STRUCT
END_TYPE

// 40 Data Types/To be Sorted/CM_CR2032_PDO_DUT
TYPE CM_CR2032_PDO_DUT :
STRUCT
	IN:CM_CR2032_PDO_IN_DUT;
	OUT:CM_CR2032_PDO_OUT_DUT;
END_STRUCT
END_TYPE

// 40 Data Types/To be Sorted/CM_CR2032_PDO_IN_DUT
TYPE CM_CR2032_PDO_IN_DUT :
STRUCT
	Digital_CH1:UINT;
	Digital_CH3:UINT;
	Digital_CH5:UINT;
	Digital_CH7:UINT;
	Analog_CH1:UINT;
	Analog_CH3:UINT;
	Analog_CH5:UINT;
	Analog_CH7:UINT;
END_STRUCT
END_TYPE

// 40 Data Types/To be Sorted/CM_CR2032_PDO_OUT_DUT
TYPE CM_CR2032_PDO_OUT_DUT :
STRUCT
	Digital:USINT;
	Analog_CH2:UINT;
	Analog_CH4:UINT;
	Analog_CH6:UINT;
	Analog_CH8:UINT;
END_STRUCT
END_TYPE

// 40 Data Types/To be Sorted/cRecipe
TYPE cRecipe :
STRUCT
	MM:cMM_Recipe;
	LTun:cLT_Recipe;
	KT:cKT_Recipe;
	WP:cWP_Recipe;
END_STRUCT
END_TYPE

// 40 Data Types/To be Sorted/eAcyclic_Response
{attribute 'qualified_only'}
//{attribute 'strict'}
TYPE eAcyclic_Response :
(
	
//Device_application_error_no_details:=16#0,
No_Error:=0,
Index_not_available:=16#11,
Subindex_not_available:=16#12,
Service_temporarily_not_available:=16#20,
Service_temporarily_NOT_available_local_control_Service:=16#21, 
temporarily_not_available_device_control:=16#22,
Access_denied:=16#23,
Parameter_value_out_OF_range:=16#30,
 
Parameter_value_above_LIMIT:=16#31,
Parameter_value_below_LIMIT :=16#32,
Parameter_length_overrun:=16#33, 
Parameter_length_underrun:=16#34,
FUNCTION_NOT_available:=16#35,
FUNCTION_temporarily_NOT_available:=16#36,

Invalid_parameter_set:=16#40,
Inconsistent_parameter_set:=16#41,
Application_NOT_ready:=16#82,





Service_NOT_available_unknown_command_has_been_sent_TO_the_IO_Link_port:=16#71,
Port_blocked_another_cyclic_process_accesses_the_IO_Link_port:=16#72,
Forbidden_access_rights_dont_allow_command_processing:=16#73,
Invalid_data_wrong_parameter_has_been_sent_in_the_command:=16#74,
Wrong_port_number:=16#76,
Wrong_port_Function_wrong_port_function_or_wrong_parameter_has_been_sent_to_the_device:=16#77,
Invalid_length_set:=16#78,
Error_in_the_device_application:=16#80


);
END_TYPE

// 40 Data Types/To be Sorted/ESL_MSG_DUT_1
TYPE ESL_MSG_DUT_1 :
STRUCT
	Device:BYTE;
	Tag:BYTE;
	Value:STRING(15);
END_STRUCT
END_TYPE

// 40 Data Types/To be Sorted/ESL_MSG_DUT
TYPE ESL_MSG_DUT :
STRUCT
	Device:BYTE;
	Tag:BYTE;
	Value:STRING(15);
END_STRUCT
END_TYPE

// 40 Data Types/To be Sorted/FIT_Transfer_DUT
TYPE FIT_Transfer_DUT :
STRUCT
	Remaining_Volume:REAL;
	Remaining_Time_S:UDINT;
	Current_Volume:REAL;
	Current_Rate:REAL;
	Status:Transfer_Status;
	Mode:FIT_Transfer_Modes;
	Config:Transfer_Config_DUT;
	
	
END_STRUCT
END_TYPE

// 40 Data Types/To be Sorted/FIT_VFD_Transfer_DUT
TYPE FIT_VFD_Transfer_DUT :
STRUCT
	Remaining_Volume:REAL;
	Remaining_Time_S:UDINT;
	Status:Transfer_Status;
	Mode:FIT_VFD_Transfer_Modes;
	Config:Transfer_Config_DUT;
	
	
END_STRUCT
END_TYPE

// 40 Data Types/To be Sorted/HSC_16Bit
TYPE HSC_16Bit :
STRUCT
	IN:HSC_Data_16Bit;
	OUT:HSC_Data_16Bit;
END_STRUCT
END_TYPE

// 40 Data Types/To be Sorted/HSC_32Bit
TYPE HSC_32Bit :
STRUCT
	IN:HSC_Data_32Bit;
	OUT:HSC_Data_32Bit;
END_STRUCT
END_TYPE

// 40 Data Types/To be Sorted/HSC_Data_16Bit
TYPE HSC_Data_16Bit :
STRUCT
	Data_Byte:BYTE;
	Data_word:WORD;
END_STRUCT
END_TYPE

// 40 Data Types/To be Sorted/HSC_Data_32Bit
TYPE HSC_Data_32Bit :
STRUCT
	Data_Byte:BYTE;
	Data_Dword:DWORD;
	
END_STRUCT
END_TYPE

// 40 Data Types/To be Sorted/HSC_DUT
TYPE HSC_DUT :
STRUCT
	Status:BYTE;
	Counter:WORD;
	Control:BYTE;
	Set_Counter_Value:WORD;
END_STRUCT
END_TYPE

// 40 Data Types/To be Sorted/Lock_DUT
TYPE Lock_DUT :
STRUCT
	Mode:INT;
	Status:INT;
	Remaining_S:INT;
	Release:BOOL;
	LED:BOOL;
	Opened:BOOL;
	
END_STRUCT
END_TYPE

// 40 Data Types/To be Sorted/Profile_DUT
TYPE Profile_DUT :
STRUCT
	Index:INT;
	Time_m:ARRAY[0..4] OF UINT;
	Target:ARRAY[0..4] OF REAL;
END_STRUCT
END_TYPE

// 40 Data Types/To be Sorted/PT_Config_DUT
TYPE PT_Config_DUT :
STRUCT
	Alarm_Config	:	Alarm_Config;
	Analog_Scale	:	Analog_scale;
	Mode			:	PT_Modes;
	
END_STRUCT
END_TYPE

// 40 Data Types/To be Sorted/Pump_PID_DUT
TYPE Pump_PID_DUT :
STRUCT
	KP:REAL;
	TN:REAL;
	TV:REAL;
	FF:REAL;
END_STRUCT
END_TYPE

// 40 Data Types/To be Sorted/Steam_Set_Config_DUT
TYPE Steam_Set_Config_DUT :
STRUCT
	Isolation_Open_Demand:REAL;
	Isolation_CLose_Demand:REAL;
	ACV_Config:cACV;
	BV_Config:cBCV;
	
	
END_STRUCT
END_TYPE

// 40 Data Types/To be Sorted/Steam_Set_DUT
TYPE Steam_Set_DUT :
STRUCT
	Mode:UINT;
	Status:UINT;
	ACV:cACV;
	BV:cBCV;
END_STRUCT
END_TYPE

// 40 Data Types/To be Sorted/Tank_Lights_DUT
TYPE Tank_Lights_DUT :
STRUCT
	CMD:BYTE;
	Status:BYTE;
	Duty:BYTE:=50;
	Output:BOOL;
	Duty_Time:TIME:=T#5M;
END_STRUCT
END_TYPE

// 40 Data Types/To be Sorted/TT_Config_DUT
TYPE TT_Config_DUT :
STRUCT
	Alarm_Config	:	Alarm_Config;
	Analog_Scale	:	Analog_scale;
	Mode			:	TT_Modes;
	
END_STRUCT
END_TYPE

// 40 Data Types/To be Sorted/Valve_3285_DUT_1
TYPE Valve_3285_DUT_1 :
STRUCT
	Mode:UINT;
	Status:UINT;
	//PDO:Valve_3285_PDO;
	PLC_SP:REAL;
	HMI_SP:REAL;
	HMI_CMD:REAL;
	Kp:REAL;
	Tv:REAL;
	Tn:REAL;
	Kp_Temp:REAL;
	Tv_Temp:REAL;
	Tn_Temp:REAL;		
END_STRUCT
END_TYPE

// 40 Data Types/To be Sorted/Valve_3285_DUT
TYPE Valve_3285_DUT :
STRUCT
	Mode:DWORD;
	Status:UINT;
	PLC_CMD:REAL;
	HMI_CMD:REAL;
	Kp:REAL;
	Tv:REAL;
	Tn:REAL;
	Kp_Temp:REAL;
	Tv_Temp:REAL;
	Tn_Temp:REAL;		
END_STRUCT
END_TYPE

// 40 Data Types/To be Sorted/Vessel_Config_Dut
TYPE Vessel_Config_Dut :
STRUCT
	MODE:INT;
	Batch_ID:INT;
	Target_Time_minutes:UINT;
	Base_SP:REAL;
	Alarms:Alarm_Config;
	DT_Rate_C_Min:REAL;
	Zone_Temp_offset:REAL:=0.5;
	
END_STRUCT
END_TYPE

// 40 Data Types/To be Sorted/Vessel_DUT
TYPE Vessel_DUT :
STRUCT
	
	//Status:INT;
	Status:BH_Vessel_Status;
	Time_Remain_S:UINT;
	Target_EU:REAL;
	Average_EU:REAL;
	Error_EU:REAL;
	Base_RCP_ID:INT;
	Loop_Index_Cone:INT;
	Loop_Index_Bottom:INT;
	Loop_Index_Middle:INT;
	Loop_Index_Top:INT;
	Config:WORD;
	
	StrMode:STRING;
	//StrTask:STRING;
	StrStatus:STRING;
END_STRUCT
END_TYPE

// 40 Data Types/To be Sorted/Vessel_PB_DUT
TYPE Vessel_PB_DUT :
STRUCT
	YL_PB:BOOL;
	YL_LED:BOOL;
	BL_PB:BOOL;
	BL_LED:BOOL;
END_STRUCT
END_TYPE

// 60 Unions/Helpers/Bytes_2_Int
TYPE Bytes_2_Int :
UNION
	Raw:ARRAY[0..1] OF BYTE;
	qInt:INT;
END_UNION
END_TYPE

// 60 Unions/Helpers/bytes_2_real
TYPE bytes_2_real :
UNION
	Raw_bytes:ARRAY[0..3] OF BYTE;
	value:REAL;
END_UNION
END_TYPE

// 60 Unions/Helpers/Bytes_DWord
TYPE Bytes_DWord :
UNION
	tByte:ARRAY[0..3] OF BYTE;
	tUSINT:ARRAY[0..3] OF USINT; 
	tInt:ARRAY[0..1] OF INT;
	tuInt:ARRAY[0..1] OF UINT;
	tWord:ARRAY[0..1] OF WORD;
	tReal:REAL;
	tDint:DINT;
	tUDINT:UDINT;
	tDword:DWORD;
	//tString:STRING(4);
	
END_UNION
END_TYPE

// 60 Unions/Helpers/Bytes_Word
TYPE Bytes_Word :
UNION
	tByte:ARRAY[0..1] OF BYTE;
	tWord: WORD;
	tInt:INT;
	tUint:UINT;
END_UNION
END_TYPE

// 60 Unions/Helpers/IFM_Status
TYPE IFM_Status :
UNION
	RX:WORD;
	Status:ARRAY[0..15] OF BOOL;
END_UNION
END_TYPE

// 60 Unions/Helpers/ORF
TYPE ORF :
UNION
	Address:DWORD;
	SDO:SDO;
END_UNION
END_TYPE

// 60 Unions/Helpers/REAL_2_WORD
TYPE REAL_2_WORD :
UNION
	rReal:REAL;
	wWord:ARRAY[0..1]OF WORD;
END_UNION
END_TYPE

// 60 Unions/Helpers/uNamur
TYPE uNamur :
UNION
	iNamur:INT;
	eNamur:eNamur107;
	
END_UNION
END_TYPE

// 60 Unions/Helpers/uUser_Confirm
TYPE uUser_Confirm :
UNION
	iConfirm:INT;
	eConfirm:eUser_Confirm;
	
END_UNION
END_TYPE

// 60 Unions/Helpers/WORD_2_Real
TYPE WORD_2_Real :
UNION
	wWord:ARRAY[0..1] OF WORD;
	rReal:REAL;
	
END_UNION
END_TYPE

// 60 Unions/Level_1/uACV_Mode
TYPE uACV_Mode :
UNION
	iMode:INT;
	eMode:eACV_Modes;
END_UNION
END_TYPE

// 60 Unions/Level_1/uACV_Status
TYPE uACV_Status :
UNION
	iStatus:INT;
	eStatus:eACV_Status;
END_UNION
END_TYPE

// 60 Unions/Level_1/uAIT_Mode
TYPE uAIT_Mode :
UNION
	iMode:INT;
	eMode:AIT_Modes;
END_UNION
END_TYPE

// 60 Unions/Level_1/uAnalog_Pump_Modes
TYPE uAnalog_Pump_Modes :
UNION
	iMode:INT;
	eMode:eAnalog_Pump_Modes;
END_UNION
END_TYPE

// 60 Unions/Level_1/uAnalog_Pump_Status
TYPE uAnalog_Pump_Status :
UNION
	iStatus:INT;
	eStatus:eAnalog_Pump_Status;
END_UNION
END_TYPE

// 60 Unions/Level_1/uBCV_Mode
TYPE uBCV_Mode :
UNION
	iMode:INT;
	eMode:eBCV_Modes;
END_UNION
END_TYPE

// 60 Unions/Level_1/uBCV_Status
TYPE uBCV_Status :
UNION
	iStatus:INT;
	eStatus:eBCV_Status;
END_UNION
END_TYPE

// 60 Unions/Level_1/uContactor_Modes
TYPE uContactor_Modes :
UNION
	iMode:INT;
	eMode:Contactor_Modes;
END_UNION
END_TYPE

// 60 Unions/Level_1/uDI_Mode
TYPE uDI_Mode :
UNION
	iMode:INT;
	eMode:DI_Modes;
END_UNION
END_TYPE

// 60 Unions/Level_1/uDI_Status
TYPE uDI_Status :
UNION
	iStatus:INT;
	eStatus:DI_Status;
END_UNION
END_TYPE

// 60 Unions/Level_1/uDo_Modes
TYPE uDo_Modes :
UNION
	iMode:INT;
	eMode:Do_modes;
END_UNION
END_TYPE

// 60 Unions/Level_1/uDuplex_mode
TYPE uDuplex_mode :
UNION
	iMode:INT;
	eMode:eDuplex_mode;
END_UNION
END_TYPE

// 60 Unions/Level_1/uHOA_Mode
TYPE uHOA_Mode :
UNION
	iMode:INT;
	eMode:eHOA_Modes;
END_UNION
END_TYPE

// 60 Unions/Level_1/uM_Pump_Modes
TYPE uM_Pump_Modes :
UNION
	iMode:INT;
	eMode:eM_Pump_Modes;
END_UNION
END_TYPE

// 60 Unions/Level_1/uM_Pump_Status
TYPE uM_Pump_Status :
UNION
	iStatus:INT;
	eStatus:eM_Pump_Status;
END_UNION
END_TYPE

// 60 Unions/Level_1/uNord_Data_In
TYPE uNord_Data_In :
UNION
	
END_UNION
END_TYPE

// 60 Unions/Level_1/uNord_Status_Word
TYPE uNord_Status_Word :
UNION
	Raw:WORD;
	Status:cNord_Status;
	
	
END_UNION
END_TYPE

// 60 Unions/Level_1/uSensor_Status
TYPE uSensor_Status :
UNION
	iStatus:INT;
	eStatus:eSensor_Status;
END_UNION
END_TYPE

// 60 Unions/Level_1/uVFD_Mode
TYPE uVFD_Mode :
UNION
	iMode:INT;
	eMode:VFD_modes;
END_UNION
END_TYPE

// 60 Unions/Level_1/uVFD_Status
TYPE uVFD_Status :
UNION
	iStatus:INT;
	eStatus:eVFD_Status;
END_UNION
END_TYPE

// 60 Unions/Level_2/uBatch_Transfer_Mode
TYPE uBatch_Transfer_Mode :
UNION
	iMode:INT;
	eMode:eBatch_Transfer_Mode;
END_UNION
END_TYPE

// 60 Unions/Level_2/uChase_Status
TYPE uChase_Status :
UNION
	iStatus:INT;
	eStatus:eChase_Status;
END_UNION
END_TYPE

// 60 Unions/Level_2/uHighSpeed_Tempered_Mode
TYPE uHighSpeed_Tempered_Mode :
UNION
	iMode:INT;
	eMode:eHighSpeed_Tempered_Mode;
END_UNION
END_TYPE

// 60 Unions/Level_2/uHighSpeed_Tempered_Status
TYPE uHighSpeed_Tempered_Status :
UNION
	iStatus:INT;
	eStatus:eHighSpeed_Tempered_Status;
END_UNION
END_TYPE

// 60 Unions/Level_2/uHighSpeed_Tempered_Task
TYPE uHighSpeed_Tempered_Task :
UNION
	iTask:INT;
	eTask:eHighSpeed_Tempered_Task;
END_UNION
END_TYPE

// 60 Unions/Level_2/uPID_Modes
TYPE uPID_Modes :
UNION
	iMode:INT;
	eMode:ePID_Modes;
	
END_UNION
END_TYPE

// 60 Unions/Level_2/uPID_Status
TYPE uPID_Status :
UNION
	iStatus:INT;
	eStatus:ePID_Status;
END_UNION
END_TYPE

// 60 Unions/Level_2/uQuick_Mix_Modes
TYPE uQuick_Mix_Modes :
UNION
	iMode:INT;
	eMode:eQuick_Mix_Modes;
END_UNION
END_TYPE

// 60 Unions/Level_2/uTempered_Modes
TYPE uTempered_Modes :
UNION
	iMode:INT;
	eMode:eTempered_Modes;
END_UNION
END_TYPE

// 60 Unions/Level_2/uTempered_Status
TYPE uTempered_Status :
UNION
	iStatus:INT;
	eStatus:eTempered_Status;
END_UNION
END_TYPE

// 60 Unions/Level_2/uTempered_Tasks
TYPE uTempered_Tasks :
UNION
	iTask:INT;
	eTask:eTempered_Task;
END_UNION
END_TYPE

// 60 Unions/Level_3/uBatch_Status
TYPE uBatch_Status :
UNION
	iStatus:INT;
	eStatus:eBatch_Status;
END_UNION
END_TYPE

// 60 Unions/Level_3/uBatch_Task
TYPE uBatch_Task :
UNION
	iTask:INT;
	eTask:eBatch_Task;
END_UNION
END_TYPE

// 60 Unions/Level_3/uBrite_Modes
TYPE uBrite_Modes :
UNION
	iMode:INT;
	eMode:eBrite_Modes;
END_UNION
END_TYPE

// 60 Unions/Level_3/uBrite_Status
TYPE uBrite_Status :
UNION
	eStatus:eBrite_Status;
	iStatus:INT;
END_UNION
END_TYPE

// 60 Unions/Level_3/uCLT_Mode
TYPE uCLT_Mode :
UNION
	iMode:INT;
	eMode:eCLT_Modes;
END_UNION
END_TYPE

// 60 Unions/Level_3/uCLT_Status
TYPE uCLT_Status :
UNION
	iStatuus:INT;
	eStatus:eCLT_Status;
END_UNION
END_TYPE

// 60 Unions/Level_3/uCLT_Task
TYPE uCLT_Task :
UNION
	iTask:INT;
	eTask:eCLT_Task;
END_UNION
END_TYPE

// 60 Unions/Level_3/uFermenter_Modes
TYPE uFermenter_Modes :
UNION
	iMode:INT;
	eMode:eFermenter_Modes;
END_UNION
END_TYPE

// 60 Unions/Level_3/uFermenter_Status
TYPE uFermenter_Status :
UNION
	eStatus:eFermenter_Status;
	iStatus:INT;
END_UNION
END_TYPE

// 60 Unions/Level_3/uFilter_Manager_Modes
TYPE uFilter_Manager_Modes :
UNION
	iMode:INT;
	eMode:eFilter_Manager_Modes;
END_UNION
END_TYPE

// 60 Unions/Level_3/uFilter_Status
TYPE uFilter_Status :
UNION
	iStatus:INT;
	eStatus:eFilter_Status;
END_UNION
END_TYPE

// 60 Unions/Level_3/uFilterMode
TYPE uFilterMode :
UNION
	iMode:INT;
	eMode:eFilter_Mode;
END_UNION
END_TYPE

// 60 Unions/Level_3/uGR_Status
TYPE uGR_Status :
UNION
	iStatuus:INT;
	eStatus:eGrain_Room_Status;
END_UNION
END_TYPE

// 60 Unions/Level_3/uGR_Task
TYPE uGR_Task :
UNION
	iTask:INT;
	eTask:eGR_Task;
END_UNION
END_TYPE

// 60 Unions/Level_3/uHLT_Mode
TYPE uHLT_Mode :
UNION
	iMode:INT;
	eMode:eHLT_Modes;
END_UNION
END_TYPE

// 60 Unions/Level_3/uHLT_Status
TYPE uHLT_Status :
UNION
	iStatuus:INT;
	eStatus:eHLT_Status;
END_UNION
END_TYPE

// 60 Unions/Level_3/uHLT_Task
TYPE uHLT_Task :
UNION
	iTask:INT;
	eTask:eHLT_Task;
END_UNION
END_TYPE

// 60 Unions/Level_3/uKT_Mode
TYPE uKT_Mode :
UNION
	iMode:INT;
	eMode:eKT_Modes;
END_UNION
END_TYPE

// 60 Unions/Level_3/uKT_Status
TYPE uKT_Status :
UNION
	iStatuus:INT;
	eStatus:eKT_Status;
END_UNION
END_TYPE

// 60 Unions/Level_3/uKT_Task
TYPE uKT_Task :
UNION
iTask:INT;
eTask:eKT_Task;
END_UNION
END_TYPE

// 60 Unions/Level_3/uLT_Mode
TYPE uLT_Mode :
UNION
	iMode:INT;
	eMode:eLT_Modes;
END_UNION
END_TYPE

// 60 Unions/Level_3/uLT_Task
TYPE uLT_Task :
UNION
iTask:INT;
eTask:eLT_Task;
END_UNION
END_TYPE

// 60 Unions/Level_3/uMM_Mode
TYPE uMM_Mode :
UNION
	iMode:INT;
	eMode:eMM_Modes;
END_UNION
END_TYPE

// 60 Unions/Level_3/uMM_Task
TYPE uMM_Task :
UNION
	iTask:INT;
	eTask:eMM_Task;
END_UNION
END_TYPE

// 60 Unions/Level_3/uWP_Mode
TYPE uWP_Mode :
UNION
	iMode:INT;
	eMode:eWP_Modes;
END_UNION
END_TYPE

// 60 Unions/Level_3/uWP_Modes
TYPE uWP_Modes :
UNION
	iMode:INT;
	eMode:eWP_Modes;
END_UNION
END_TYPE

// 60 Unions/Level_3/uWP_Status
TYPE uWP_Status :
UNION
	iStatus:INT;
	eStatus:eWP_Status;
END_UNION
END_TYPE

// 60 Unions/Level_3/uWP_Task
TYPE uWP_Task :
UNION
	iTask:INT;
	eTask:eWP_Task;
END_UNION
END_TYPE

// 70 Modes Enums/Brewery/BH_Vessel_Modes
{attribute 'qualified_only'}
{attribute 'strict'}
TYPE BH_Vessel_Modes :
(
	Off:=0,
	Zones_Equal,
	Top_Cold,
	Bottom_Cold,
	Top_Only,
	Middle_Only,
	Bottom_Only,
	Cone_Only
	
);
END_TYPE

// 70 Modes Enums/Brewery/CIP_1_Modes
{attribute 'qualified_only'}
//{attribute 'strict'}
TYPE CIP_1_Modes :
(
	Off := 0,
	Auto_Run,
	Auto_Paused,
	Auto_Halt
	
);
END_TYPE

// 70 Modes Enums/Brewery/eBrite_Modes
{attribute 'qualified_only'}
//{attribute 'strict'}
{attribute 'to_string'}
TYPE eBrite_Modes :
(
	Off := 0,
	ON//,
	//Crash
);
END_TYPE

// 70 Modes Enums/Brewery/eCLT_Modes
{attribute 'qualified_only'}
//{attribute 'strict'}
{attribute 'to_string'}
TYPE eCLT_Modes :
(
	Off := 0,
	Auto,
	Manual
	
);
END_TYPE

// 70 Modes Enums/Brewery/eFermenter_Modes
{attribute 'qualified_only'}
//{attribute 'strict'}
{attribute 'to_string'}
TYPE eFermenter_Modes :
(
	Off := 0,
	Ferment,
	Crash
);
END_TYPE

// 70 Modes Enums/Brewery/eGR_Modes
{attribute 'qualified_only'}
//{attribute 'strict'}
{attribute 'to_string'}
TYPE eGR_Modes :
(
	Off := 0,
	Mill,
	Transfer,
	Auto_Halt
	
);
END_TYPE

// 70 Modes Enums/Brewery/eHLT_Modes
{attribute 'qualified_only'}
//{attribute 'strict'}
{attribute 'to_string'}
TYPE eHLT_Modes :
(
	Off := 0,
	Auto,
	Manual
	
);
END_TYPE

// 70 Modes Enums/Brewery/eKT_Mode
TYPE eKT_Mode :
UNION
	iMode:INT;
	eMode:eKT_Modes;
END_UNION
END_TYPE

// 70 Modes Enums/Brewery/eLT_Modes
{attribute 'qualified_only'}
//{attribute 'strict'}
{attribute 'to_string'}
TYPE eLT_Modes :
(
	Off := 0,
	Auto,
	Manual,
	Pause
	
);
END_TYPE

// 70 Modes Enums/Brewery/eMM_Modes
{attribute 'qualified_only'}
//{attribute 'strict'}
{attribute 'to_string'}
TYPE eMM_Modes :
(
	Off := 0,
	Auto,
	Manual
);
END_TYPE

// 70 Modes Enums/Brewery/FV_Modes
{attribute 'qualified_only'}
//{attribute 'strict'}
TYPE FV_Modes :
(
	Off := 0,
	Ferment,
	Dry_Hop,
	Crash
	
);
END_TYPE

// 70 Modes Enums/Brewery/HLT_Blending_Modes
{attribute 'qualified_only'}
//{attribute 'strict'}
TYPE HLT_Blending_Modes :
(
	Off := 0,
	Auto_Run,
	Auto_Paused,
	Auto_Halt
	
);
END_TYPE

// 70 Modes Enums/Brewery/KTWP_Modes
{attribute 'qualified_only'}
//{attribute 'strict'}
{attribute 'to_string'}
TYPE KTWP_Modes :
(
	Off := 0,
	Auto_Run,
	Auto_Paused,
	Auto_Halt
	
);
END_TYPE

// 70 Modes Enums/Brewery/MM_Decoction_Modes
{attribute 'qualified_only'}
//{attribute 'strict'}
TYPE MM_Decoction_Modes :
(
	Off := 0,
	Auto_Run,
	Auto_Paused,
	Auto_Halt
	
);
END_TYPE

// 70 Modes Enums/Level_0/eMB0_RTD_Input_Type
{attribute 'qualified_only'}
{attribute 'strict'}
TYPE eMB0_RTD_Input_Type :
(
	Disabled := 0,
	R0_200:=16#0012,
	R0_500:=16#000C,
	Pt100:=16#000D,
	Ni100:=16#000F,
	PT1000:=16#000E,
	Ni1000:=16#0010,
	Pot_50k:=16#11
);
END_TYPE

// 70 Modes Enums/Level_0/eMB0_RTD_Units
{attribute 'qualified_only'}
{attribute 'strict'}
TYPE eMB0_RTD_Units :
(
	C := 0,
	F:=16#0001,
	K:=16#0002
);
END_TYPE

// 70 Modes Enums/Level_0/Reset_Relay_Mode
{attribute 'qualified_only'}
{attribute 'strict'}
TYPE Reset_Relay_Mode :
(
	Off := 0,
	On
	
);
END_TYPE

// 70 Modes Enums/Level_1/AIT_Modes
{attribute 'qualified_only'}
//{attribute 'strict'}
{attribute 'to_string'}
TYPE AIT_Modes :
(
	Active := 0,
	Forced,
	Alarms_Disabled,
	Alarm_Reset,
	OffLine
);
END_TYPE

// 70 Modes Enums/Level_1/Command_Modes
{attribute 'qualified_only'}
//{attribute 'strict'}
TYPE Command_Modes :
(
	Off := 0,
	Auto_Run,
	Auto_Paused,
	Auto_Complete,
	Auto_Halt
	
);
END_TYPE

// 70 Modes Enums/Level_1/Contactor_Modes
{attribute 'qualified_only'}
{attribute 'to_string'}
TYPE Contactor_Modes :
(
	Auto := 0,
	Fwd,
	Bump_FWD,
	Disabled,
	Rev,
	Bump_REV
);
END_TYPE

// 70 Modes Enums/Level_1/Di_Modes
{attribute 'qualified_only'}
{attribute 'strict'}
{attribute 'to_string'}
TYPE Di_Modes :
(
	Auto := 0,
	Forced_On,
	Forced_Off
);
END_TYPE

// 70 Modes Enums/Level_1/DO_Modes
{attribute 'qualified_only'}
//{attribute 'strict'}
{attribute 'to_string'}
TYPE DO_Modes :
(
	Auto := 0,
	Forced_Off,
	Forced_On
);
END_TYPE

// 70 Modes Enums/Level_1/e_8681_Modes
{attribute 'qualified_only'}
//{attribute 'strict'}
TYPE e_8681_Modes :
(
	Auto := 0,
	Disabled,
	Open,
	Upper_Drain,
	Lower_Drain
);
END_TYPE

// 70 Modes Enums/Level_1/eACV_Modes
{attribute 'qualified_only'}
//{attribute 'strict'}
{attribute 'to_string'}
TYPE eACV_Modes :
(
	Auto := 0,
	Closed,
	Open,
	Locate,
	xTune,
	Burkert_Open,//5
	Manual_Pos,
	Simulate
	
	
);
END_TYPE

// 70 Modes Enums/Level_1/eAnalog_Control_Modes
{attribute 'qualified_only'}
//{attribute 'strict'}
{attribute 'to_string'}
TYPE eAnalog_Control_Modes :
(
	Auto := 0,
	OFF,
	Manual
);
END_TYPE

// 70 Modes Enums/Level_1/eAnalog_Pump_Modes
{attribute 'qualified_only'}
//{attribute 'strict'}
{attribute 'to_string'}
TYPE eAnalog_Pump_Modes :
(
	Auto := 0,
	Disabled,
	Manual,
	Prime,
	Calibrate
	
);
END_TYPE

// 70 Modes Enums/Level_1/eAODD_Modes
{attribute 'qualified_only'}
//{attribute 'strict'}
{attribute 'to_string'}
TYPE eAODD_Modes :
(
	Auto := 0,
	Disabled,
	Manual,
	Prime
);
END_TYPE

// 70 Modes Enums/Level_1/eB336x_Modes
{attribute 'qualified_only'}
//{attribute 'strict'}
TYPE eB336x_Modes :
(
		Auto := 0,
	Closed,
	Open,
	Manual_Pos,
	Config
);
END_TYPE

// 70 Modes Enums/Level_1/eBCV_Modes
{attribute 'qualified_only'}
//{attribute 'strict'}
{attribute 'to_string'}

TYPE eBCV_Modes :
(
	Auto:=0,
	Closed,
	Open,
	Identify,
	xTune,
	Burkert_Open, //5
	Simulate:=7
	
);
END_TYPE

// 70 Modes Enums/Level_1/eConfig_startTune
{attribute 'qualified_only'}
//{attribute 'strict'}
TYPE eConfig_startTune :
(
	Complete := 0,
	Abort:=1,
	x_Tune:=2,
	p_Tune:=3,
	p_Lin:=4,
	a_Tune:=5,
	m_Clean:=7,
	mQC:=9
);
END_TYPE

// 70 Modes Enums/Level_1/eHOA_Modes
{attribute 'qualified_only'}
//{attribute 'strict'}
{attribute 'to_string'}
TYPE eHOA_Modes :
(
	Auto := 0,
	Off,
	Manual
);
END_TYPE

// 70 Modes Enums/Level_1/eM_Pump_Modes
{attribute 'qualified_only'}
{attribute 'strict'}
{attribute 'to_string'}
TYPE eM_Pump_Modes :
(
	Auto := 0,
	Disbaled,
	Manual,
	Prime,
	Calibrate
	
);
END_TYPE

// 70 Modes Enums/Level_1/Fan_Modes
{attribute 'qualified_only'}
//{attribute 'strict'}
TYPE Fan_Modes :
(
	Off := 0,
	On,
	Auto
	
);
END_TYPE

// 70 Modes Enums/Level_1/LS_Modes
{attribute 'qualified_only'}
{attribute 'strict'}
TYPE LS_Modes :
(
	Active := 0,
	Forced_Off,
	Forced_On
);
END_TYPE

// 70 Modes Enums/Level_1/Positioner_Modes
{attribute 'qualified_only'}
{attribute 'strict'}
TYPE Positioner_Modes :
(
	Auto := 0,
	Manual_Open,
	Manual_Close,
	Manual_Position
);
END_TYPE

// 70 Modes Enums/Level_1/PT_Modes
{attribute 'qualified_only'}
//{attribute 'strict'}
TYPE PT_Modes :
(
	Active := 0,
	Forced,
	Alarms_Disabled,
	Alarm_Reset,
	OffLine
);
END_TYPE

// 70 Modes Enums/Level_1/TT_Modes
{attribute 'qualified_only'}
//{attribute 'strict'}
TYPE TT_Modes :
(
	Active := 0,
	Forced,
	Alarms_Disabled,
	Alarm_Reset,
	OffLine
);
END_TYPE

// 70 Modes Enums/Level_1/VFD_Modes
{attribute 'qualified_only'}
//{attribute 'strict'}
{attribute 'to_string'}
TYPE VFD_Modes :
(
	Auto := 0,
	Disabled,
	Manual,
	Reset,
	Simulate:=10
);
END_TYPE

// 70 Modes Enums/Level_2/AIT_Transfer_Modes
{attribute 'qualified_only'}
//{attribute 'strict'}
TYPE AIT_Transfer_Modes :
(
	Idle := 0,
	Maintain_Target,
	//Flow_Only,
	Hz_only,
	//Pressure_Only,
	//LS_Dry,
	//Flow_Timed,
	Timed,
	Hz_Timed,
	//Pressure_Timed,
	//Batch,
	Lock_Out,
	Passive,
	Pause,
	Resume
	);
END_TYPE

// 70 Modes Enums/Level_2/eBatch_Transfer_Mode
{attribute 'qualified_only'}
//{attribute 'strict'}
{attribute 'to_string'}
TYPE eBatch_Transfer_Mode :
(
	Auto := 0,
	Batch,
	Disabled,
	Pause,
	Resume
	);
END_TYPE

// 70 Modes Enums/Level_2/eChase_Mode
{attribute 'qualified_only'}
//{attribute 'strict'}
{attribute 'to_string'}
TYPE eChase_Mode :
(
	Auto := 0,
	OFF,
	Manual
);
END_TYPE

// 70 Modes Enums/Level_2/eDuplex_Mode
{attribute 'qualified_only'}
{attribute 'strict'}
TYPE eDuplex_Mode :
(
	Auto := 0,
	Force_1,
	Force_2,
	Disabled
);
END_TYPE

// 70 Modes Enums/Level_2/eFilter_Manager_Modes
{attribute 'qualified_only'}
{attribute 'strict'}
TYPE eFilter_Manager_Modes :
(
	Auto := 0,
	Filter_1,
	Filter_2,
	Disabled,
	Bypass,
	Manual
);
END_TYPE

// 70 Modes Enums/Level_2/eFilter_Mode
{attribute 'qualified_only'}
{attribute 'to_string'}
TYPE eFilter_Mode :
(
	Idle := 0,
	Prime,
	Active,
	Drain,
	Rinse,
	Disabled:=10,		//10
	Maintenance	//11
);
END_TYPE

// 70 Modes Enums/Level_2/eHighSpeed_Tempered_Mode
{attribute 'qualified_only'}
{attribute 'strict'}
TYPE eHighSpeed_Tempered_Mode :
(
	OFF := 0,
	Manual,
	Auto
);
END_TYPE

// 70 Modes Enums/Level_2/ePID_Modes
{attribute 'qualified_only'}
//{attribute 'strict'}
{attribute 'to_string'}
TYPE ePID_Modes :
(
	Auto := 0,
	FORCED_OFF,
	FORCED_ON	
);
END_TYPE

// 70 Modes Enums/Level_2/eQuick_Mix_Modes
{attribute 'qualified_only'}
//{attribute 'strict'}
{attribute 'to_string'}
TYPE eQuick_Mix_Modes :
(
	Auto := 0,
	OFF,
	Manual,
	Pause
);
END_TYPE

// 70 Modes Enums/Level_2/eTempered_Modes
{attribute 'qualified_only'}
//{attribute 'strict'}
{attribute 'to_string'}
TYPE eTempered_Modes :
(
	Auto:=0,
	OFF,
	Manual
);
END_TYPE

// 70 Modes Enums/Level_2/FIT_Transfer_Modes
{attribute 'qualified_only'}
//{attribute 'strict'}
TYPE FIT_Transfer_Modes :
(
	Idle := 0,
	//AIT_Only,
	//Flow,
	//Hz_only,
	//Pressure_Only,
	//LS_Dry,
	//Flow_Timed,
	//AIT_Timed,
	//Hz_Timed,
	//Pressure_Timed,
	Batch,
	Lock_Out,
	Passive,
	Pause,
	Resume
	);
END_TYPE

// 70 Modes Enums/Level_2/FIT_VFD_Transfer_Modes
{attribute 'qualified_only'}
//{attribute 'strict'}
TYPE FIT_VFD_Transfer_Modes :
(
	Idle := 0,
	//AIT_Only,
	//Flow_Only,
	//Hz_only,
	//Pressure_Only,
	//LS_Dry,
	//Flow_Timed,
	//AIT_Timed,
	//Hz_Timed,
	//Pressure_Timed,
	Batch,
	Lock_Out,
	Passive,
	Pause,
	Resume
	);
END_TYPE

// 70 Modes Enums/Level_2/Mix_Modes
{attribute 'qualified_only'}
{attribute 'to_string'}
//{attribute 'strict'}

TYPE Mix_Modes :
(
	Idle := 0,
	Pause,
	Resume,
	Auto,
	Quick_Start, //Skips Foundation Control and start testing.
	Endless, // Target Volume is Ignored
	Rate_Only,
	Temperature_Only,
	Hot_Only,
	Cold_Only
	
	
	
);
END_TYPE

// 70 Modes Enums/Level_2/Steam_Condensate_Modes
{attribute 'qualified_only'}
//{attribute 'strict'}
TYPE Steam_Condensate_Modes :
(
	Ready := 0,
	Condensdate_Return
	
);
END_TYPE

// 70 Modes Enums/Level_2/Steam_Modes
{attribute 'qualified_only'}
//{attribute 'strict'}
TYPE Steam_Modes :
(
	Off := 0,
	Blow_Down,
	Ready
	
);
END_TYPE

// 70 Modes Enums/Level_2/Temp_loop_Modes
{attribute 'qualified_only'}
//{attribute 'strict'}
TYPE Temp_loop_Modes :
(
	Idle := 0,
	Crash,
	Profile,
	Step,
	Auto,
	Auto_Paused
);
END_TYPE

// 70 Modes Enums/Level_3/CLT_Modes
{attribute 'qualified_only'}
//{attribute 'strict'}
TYPE CLT_Modes :
(
	Off := 0,
	Auto_Run,
	Auto_Paused,
	Auto_Halt
	
);
END_TYPE

// 70 Modes Enums/Level_3/eKT_Modes
{attribute 'qualified_only'}
//{attribute 'strict'}
{attribute 'to_string'}
TYPE eKT_Modes :
(
	Auto := 0,
	OFF,
	Manual
);
END_TYPE

// 70 Modes Enums/Level_3/eRCP_Mode
{attribute 'qualified_only'}
//{attribute 'strict'}
TYPE eRCP_Mode :
(
	Ready:= 0,
	Activate,
	Save,
	Copy,
	Paste,
	ReLoad,
	Push_To_MT,
	Push_To_LT,
	Push_To_KT,
	Push_To_WP,
	Pull_From_MT,
	Pull_From_LT,
	Pull_From_KT,
	Pull_From_WP
	
);
END_TYPE

// 70 Modes Enums/Level_3/eWP_Modes
{attribute 'qualified_only'}
//{attribute 'strict'}
{attribute 'to_string'}
TYPE eWP_Modes :
(
	Auto := 0,
	OFF,
	Manual
);
END_TYPE

// 80 Status Enums/Level_0/eNamur107
{attribute 'qualified_only'}
//{attribute 'strict'}
{attribute 'to_string'}
TYPE eNamur107 :
(
	Normal := 0,			//White
	OK,						//Green
	MaintenanceReq,			//Blue
	OutOfSpec,				//Yellow
	Warning,				//Orange
	Error,					//Red
	
	Offline:=10				//black
	
);
END_TYPE

// 80 Status Enums/Level_0/eORF_Status
{attribute 'qualified_only'}
//{attribute 'strict'}
TYPE eORF_Status :
(
	NoError:=16#00,
	GeneralError:=16#02,
	No_Subindex_specifed:=16#04,
	Access_NOT_supported:=16#05,
	Data_length_too_great:=16#09,
	Data_length_too_small:=16#0A,
	No_object:=16#0F,
	Service_could_not_be_implemented:=16#11,
	Read_access_only:=16#1F,
	No_data:=16#21,
	No_device_with_this_Node_ID_available:=16#FF,
	Processisrunning:=16#FFFF
);
END_TYPE

// 80 Status Enums/Level_0/SDO_Error_Codes
{attribute 'qualified_only'}
{attribute 'strict'}
TYPE SDO_Error_Codes :
	(
	Dummy:=0
(*
	 SDO_ERR_TOGGLE_BIT   :=16#05030000,
 
 	SDO_ERR_TIMEOUT   :=16#05040000,
 
 	SDO_ERR_COMMAND   :=16#05040001,
 
 	SDO_ERR_BLOCK_SIZE   :=16#05040002,
 
 	SDO_ERR_BLOCK_SEQUENCE   :=16#05040003,
 
 	SDO_ERR_BLOCK_CRC   :=16#05040004,
 
 	SDO_ERR_MEMORY   :=16#05040005,
 
 	SDO_ERR_ACCESS_UNSUPPORTED   :=16#06010000,
 
 	SDO_ERR_ACCESS_WO   :=16#06010001,
 
 	SDO_ERR_ACCESS_RO   :=16#06010002
 
 	SDO_ERR_NO_OBJECT   :=16#06020000
 
 	SDO_ERR_MAPPING_OBJECT   :=16#06040041
 
 	SDO_ERR_MAPPING_LENGTH   :=16#06040042
 
 	SDO_ERR_GENERAL_PARAMETER   :=16#06040043
 
 	SDO_ERR_GENERAL_DEVICE   :=16#06040047
 
 	SDO_ERR_HARDWARE   :=16#06060000
 
 	SDO_ERR_DATATYPE   :=16#06070010
 
 	SDO_ERR_DATATYPE_HIGH   :=16#06070012
 
 	SDO_ERR_DATATYPE_LOW   :=16#06070013
 
 	SDO_ERR_NO_SUB_INDEX   :=16#06090011
 
 	SDO_ERR_VALUE_RANGE   :=16#06090030
 
 	SDO_ERR_VALUE_HIGH   :=16#06090031
 
 	SDO_ERR_VALUE_LOW   :=16#06090032
 
 	SDO_ERR_VALUE_MIN_MAX   :=16#06090036
 
 	SDO_ERR_SDO_CONNECTION   :=16#060A0023
 
 	SDO_ERR_GENERAL   :=16#08000000
 
 	SDO_ERR_DATA_STORE   :=16#08000020
 
 	SDO_ERR_DATA_STORE_LOCAL   :=16#08000021
 
 	SDO_ERR_DATA_STORE_STATE   :=16#08000022
 
 	SDO_ERR_OBJECT_DICTIONARY   :=16#08000023
 
 	SDO_ERR_NO_DATA   :=16#08000024
*)
);
END_TYPE

// 80 Status Enums/Level_1/Contactor_Status
{attribute 'qualified_only'}
{attribute 'to_string'}
TYPE Contactor_Status :
(
	OFF := 0,
	Auto_FWD,
	Auto_Rev,
	Manual_FWD,
	Manual_Rev,
	FWD_Limit,
	REV_Limit
);
END_TYPE

// 80 Status Enums/Level_1/DI_Status
{attribute 'qualified_only'}
//{attribute 'strict'}
{attribute 'to_string'}
TYPE DI_Status :
(
	Normal_Signal_OFF := 0,
	Normal_Signal_Active,
	ALARM_Signal_ACTIVE,
	ALARM_Signal_LOST,		//3
	Forced_On,
	Forced_OFF,
	Liquid_Detected,		//6
	No_Liquid_Detected,		//7
	Liquid_Detected_Alarm,	//8
	No_Liquid_Detected_Alarm,	//9
	IO_Fault,
	
	End_Status:=99
);
END_TYPE

// 80 Status Enums/Level_1/DO_Status
{attribute 'qualified_only'}
//{attribute 'strict'}
{attribute 'to_string'}
TYPE DO_Status :
(
	OFF := 0,
	On,
	Forced_OFF,
	Forced_ON,
	
	LOCKED_OUT:=6,
	Interlocked,
	OFFLINE
);
END_TYPE

// 80 Status Enums/Level_1/e8691_ValveMode
{attribute 'qualified_only'}
//{attribute 'strict'}
{attribute 'to_string'}
TYPE e8691_ValveMode :
(

	Init:=0,
	Normal,
	Tune,
	Safe
	
);
END_TYPE

// 80 Status Enums/Level_1/e8691_xTuneStatus
{attribute 'qualified_only'}
//{attribute 'strict'}
{attribute 'to_string'}
TYPE e8691_xTuneStatus :
(
	Ready:=0,
	Init,
	POS1,
	POS2,
	Stroke,
	SwTimes,
	
	errAbort:=250,
	errSafePos:=251,
	errSwTimes:=252,
	errStroke:=253,
	errPos2:=254,
	errPos1:=255
);	
END_TYPE

// 80 Status Enums/Level_1/e8694_xTuneStatus
{attribute 'qualified_only'}
//{attribute 'strict'}
{attribute 'to_string'}
TYPE e8694_xTuneStatus :
(
	Complete := 0,
	Ready,
	Init,
	EndStops,
	Leakage,
	Offset,
	Friction,
	Controller,
	NeverRan:=127,
	errTurnPoti:=250,
	errLeakageYB:=251,
	errLeakage:=252,
	errTimeOut:=253,
	errBreakErr:=254,
	errBreakUser:=255
);	
END_TYPE

// 80 Status Enums/Level_1/eACV_Status
{attribute 'qualified_only'}
//{attribute 'strict'}
{attribute 'to_string'}

TYPE eACV_Status :
(
	A_Closed:=0,
	A_Open,
	M_Closed,
	M_Open,
	Opening, //
	Closing, //
	
	LOCKED_OUT,		//6
	Interlocked,	//
	OFFLINE,		//8
	
	Fault,		//9
	Pos_Error,
	Error,// Namur 5	-,
		
		//
	Missing,		//12
	Detected,
	P_Fault,
	Maintenance_Required,//Namur  2  
	Out_Of_Spec, //Namur 3	-
	Check_Function,//Namur 4	-
	Not_Used_Manual,
	A_Position,			//19
	M_Position,			//20
	Active,				//21
	Positon_Hold		//22
				//
);
END_TYPE

// 80 Status Enums/Level_1/eAnalog_Pump_Status
{attribute 'qualified_only'}
//{attribute 'strict'}
{attribute 'to_string'}
TYPE eAnalog_Pump_Status :
(
	IDLE := 0,
	Running,
	Disabled,
	Prime,
	Manual,
	Complete,
	LOCKED_OUT,				//
	Interlocked,		//
	Offline,
	Pump_Fault,
	Fault//
);
END_TYPE

// 80 Status Enums/Level_1/eAODD_Status
{attribute 'qualified_only'}
//{attribute 'strict'}
TYPE eAODD_Status :
(
	Idle:=0,
	Disabled,
	Active,
	Complete
);
END_TYPE

// 80 Status Enums/Level_1/eB8681_Status
{attribute 'qualified_only'}
//{attribute 'strict'}
TYPE eB8681_Status :
(	
	Unknown:=0,
	Blocked,
	Open,
	Upper_Drain,
	Lower_Drain,
	Missing,
	Detected,
	P_Fault
);
END_TYPE

// 80 Status Enums/Level_1/eBCV_Status
{attribute 'qualified_only'}
//{attribute 'strict'}
{attribute 'to_string'}

TYPE eBCV_Status :
(
	A_Closed := 0,
	A_Open,			//1
	M_Closed,
	M_Open,			//3
	Opening,
	Closing,//5
	LOCKED_OUT:=6,
	Interlocked,
	OFFLINE,
	
	Fault,		//9
	Both_Limits_Active,
	Error,// Namur 5
	
	Missing,	//12
	Detected,
	P_Fault,
	Maintenance_Required,//Namur  2  -15
	Out_Of_Spec, //Namur 3	-16
	Check_Function,//Namur 4	-17,
	Failed_To_Open,			//18
	Failed_To_Close,		//19
	No_Limits_Active,		//20
	
	Status99:=99

	
);
END_TYPE

// 80 Status Enums/Level_1/eCurrentOpMode
{attribute 'qualified_only'}
//{attribute 'strict'}
{attribute 'to_string'}
TYPE eCurrentOpMode :
(
	xControl := 1,
	CutOffUp,
	CutOffDn,
	SafePosUp,
	SafePosDn,
	SafePos,
	Manual,
	xTune
	
);
END_TYPE

// 80 Status Enums/Level_1/eFloWave_Status
{attribute 'qualified_only'}
//{attribute 'strict'}
TYPE eFloWave_Status :
(
	OK := 0,
	General_Device_Alarm,
	OffLine,
	High_High_Alarm,
	High_Warning,
	Low_Warning,
	Low_Low_Alarm
	
);
END_TYPE

// 80 Status Enums/Level_1/eM_Pump_Status
{attribute 'qualified_only'}
{attribute 'strict'}
{attribute 'to_string'}
TYPE eM_Pump_Status :
(
	Idle := 0,
	Active,
	Disabled,
	Manual_Run,
	Prime_Active,
	
	
	LOCKED_OUT:=6,				//
	Interlocked,		//
	Offline
	
);
END_TYPE

// 80 Status Enums/Level_1/eSensor_Status
{attribute 'qualified_only'}
//{attribute 'strict'}
{attribute 'to_string'}
TYPE eSensor_Status :
(
	OK := 0,
	Low_Low_Alarm,	//1
	Low_Warning,	//2
	High_Warning,	//3
	HiHi_Alarm,		//4
	Offline, 
	FORCED,
	Alarms_Disabled,	//7
	Under_Range,
	Over_Range,
	Missing,
	Detected,
	P_Fault,
	Fault,
	Low_Norm,		//14
	High_Norm
);
END_TYPE

// 80 Status Enums/Level_1/eVFD_Status
{attribute 'qualified_only'}
//{attribute 'strict'}
{attribute 'to_string'}
TYPE eVFD_Status :
(
	READY:=0,	
	A_Running,				//
	Disabled,				//	
	M_Runing:=4,					//
	Ramping,				//			
			

				
	LOCKED_OUT:=6,				//
	Interlocked,		//
	Offline,
	Fault,
	Low_Voltage,  //10
	Safe_Torque_Off,
	No_Motor_Load_Detected,		//	12
	Low_Low_Current_Alarm,		//13		Sensor:1
	Low_Current_Warning,				//	Sensor:2
	High_Current_Warning,
	High_High_Current_Alarm			//	16
);
END_TYPE

// 80 Status Enums/Level_1/Positioner_Status
{attribute 'qualified_only'}
//{attribute 'strict'}
TYPE Positioner_Status :
(
	Locked_OUT := 0,
	Open,
	Closed,
	Manual
);
END_TYPE

// 80 Status Enums/Level_1/PT_Status
{attribute 'qualified_only'}
//{attribute 'strict'}
TYPE PT_Status :
(
	OK := 0,
	Low_Warning,
	Low_Low_Alarm,
	High_Warning,
	HiHi_Alarm,
	Offline,
	BurnOut,
	FORCED
	
);
END_TYPE

// 80 Status Enums/Level_1/SV_Status
{attribute 'qualified_only'}
//{attribute 'strict'}
{attribute 'to_string'}
TYPE SV_Status :
(
	Closed := 0,
	Open,
	Manual_Closed,
	Manual_Open,
	LOCKED_OUT,
	Permisive_OFF
);
END_TYPE

// 80 Status Enums/Level_1/TT_Status
{attribute 'qualified_only'}
//{attribute 'strict'}
TYPE TT_Status :
(
	OK := 0,
	Low_Warning,
	Low_Low_Alarm,
	High_Warning,
	HiHi_Alarm,
	Offline,
	BurnOut,
	FORCED
	
);
END_TYPE

// 80 Status Enums/Level_1/VFD_Fault_Status
{attribute 'qualified_only'}
//{attribute 'strict'}
{attribute 'to_string'}
TYPE VFD_Fault_Status :
(
	enum_member := 0,
	Motor_Temperature:=16
	
);
END_TYPE

// 80 Status Enums/Level_2/eChase_Status
{attribute 'qualified_only'}
//{attribute 'strict'}
{attribute 'to_string'}
TYPE eChase_Status :
(
	IDLE := 0,
	System_Stop,
	FIT_Reset,
	Active,
	Complete,
	Source_Not_Ready,
	Destination_Not_Ready,
	Not_Available,
	Open_Valve
);
END_TYPE

// 80 Status Enums/Level_2/eCondensate_Status
{attribute 'qualified_only'}
{attribute 'to_string'}
TYPE eCondensate_Status :
(
	IDLE := 0,
	Stage_1,
	Stage_2,
	High_Warning,
	HIGH_Alarm,
	Level_Switch_Fault,
	Fault
	
);
END_TYPE

// 80 Status Enums/Level_2/eFilter_Manager_Status
{attribute 'qualified_only'}
//{attribute 'strict'}
{attribute 'to_string'}
TYPE eFilter_Manager_Status :
(
	Idle := 0,
	Enable_Filter_1,
	Enable_Filter_2,
	Filter_1_Active,
	Filter_1_Only,
	Filter_1_Manual,
	Filter_1_x_2,
	Filter_2_Active,
	Filter_2_Only,
	Filter_2_Manual,
	Filter_2_x_1,
	
	No_Filter_Available,
	Disabled,
	Bypassed,
	Manual

);
END_TYPE

// 80 Status Enums/Level_2/eFilter_Status
{attribute 'qualified_only'}
{attribute 'to_string'}
TYPE eFilter_Status :
(
	IDLE := 0,
	In_Service,
	Backwash_Active,
	Prime_Active,
	Drain_Active,
	Drain_Complete,
	Pressure_Warning,
	Pressure_Alarm,
	Maintenance_Required,
	
	Prime_Complete,
	Prime_Required,
	Backwash_Complete,
	
	Open_Inlet,
	Open_Outlet,
	Close_Inlet,
	Close_Outlet,

	Open_Vent,
	Open_Drain,
	Open_Backwash,
	
	
	Valves_Not_Ready,
	Pressure_Not_Ready,
	Disabled,
	Filter_Empty,
	Bypassed
);
END_TYPE

// 80 Status Enums/Level_2/eHighSpeed_Tempered_Status
{attribute 'qualified_only'}
{attribute 'strict'}
TYPE eHighSpeed_Tempered_Status :
(
	OFF := 0,
	Calibrate_Max_Flow,
	Calibrate_2,
	Calibrate_3,
	Calibrate_4,
	Calibrate_5,
	Calibrate_6,
	Calibrate_7,
	Calibrate_8,
	Calibrate_9,
	Calibrate_10,
	Calibrate_11,
	Calibrate_12,
	Calibrate_13,
	Calibrate_14,
	Calibrate_15,
	Calibrate_16,
	Calibrate_17,
	Calibrate_18,
	Calibrate_19,
	Calibrate_20,
	Calibrate_21,
	Calibrate_22,
	Calibrate_23,
	Calibrate_24,
	Calibrate_Complete,
	
	Manual_Run,
	Auto_Run,
	Start,
	OK,
	
	High_Warning,
	Low_Waring,
	High_Alarm,
	Low_Alarm
	
);
END_TYPE

// 80 Status Enums/Level_2/ePID_Status
{attribute 'qualified_only'}
//{attribute 'strict'}
{attribute 'to_string'}
TYPE ePID_Status :
(
	Disabled := 0,
	Ready,
	Active,
	CV_Not_Ready,
	PV_Not_Ready,
	Interlocked:=7,
	Forced_ON
);
END_TYPE

// 80 Status Enums/Level_2/eQuick_Mix_Status
{attribute 'qualified_only'}
//{attribute 'strict'}
{attribute 'to_string'}
TYPE eQuick_Mix_Status :
(
	IDLE := 0,
	Fit_Reset,
	Start_Flow,
	Flow_Detected,
	Start_temperature, //4
	Temperature_OK,
	Foundation_Rate,
	Foundation_Rate_OK,		//7
	Foundation_Amount_Complete, //
	Main_Rate,
	Main_Rate_OK,//10
	Grain_Dispense,	//11
	Batch_Ending,
	Batch_Complete,
	Rate_Fault,//14
	Temperature_Fault,
	HW_Valve_Not_Ready,
	CW_Valve_Not_Ready,
	Pump_Not_Ready,
	
	Systems_Test,
	HW_Not_Ready,
	CW_Not_Ready,
	Flow_Not_Ready,
	TT_Not_Ready,//23
	On_Target,//24
	Flow_Warning, //25
	Flow_Fault,
	Temp_Warning,//27
	Temp_Fault,
	Paused,  //29
	Destination_Not_Ready//30
	
);
END_TYPE

// 80 Status Enums/Level_2/eTempered_Status
{attribute 'qualified_only'}
//{attribute 'strict'}
{attribute 'to_string'}
TYPE eTempered_Status :
(
	OFF := 0,
	Starting,
	Ready,
	Active,
	Traget_1_Machine,
	Target_2_Machines,
	Target_3_Machines,
	Target_4_Machines,
	
	Calibrating_Flow,
	Flow_On_Target,
	Adjusting_Hardness,
	Hardness_On_Target,
	
	Draining,
	Drain_Complete,
	
	Rinse_Active,
	Rinse_Complete,
	
	Prepare_Standby,
	Prepare_Active,
	Prepare_Complete,
	Prime_Start,
	Prime_Active,
	Prime_Complete,
	
	Fault
);
END_TYPE

// 80 Status Enums/Level_2/Mix_Status
{attribute 'qualified_only'}
//{attribute 'strict'}
{attribute 'to_string'}
TYPE Mix_Status :
(
	IDle := 0,
	Fit_Reset,
	Start_Flow,
	Flow_Detected,
	Start_temperature, //4
	Temperature_OK,
	Foundation_Rate,
	Foundation_Rate_OK,
	Foundation_Amount_Complete,
	Main_Rate,
	Main_Rate_OK,//10
	Grain_Dispense,
	Batch_Ending,
	Batch_Complete,
	Rate_Fault,
	Temperature_Fault,
	HW_Valve_Not_Ready,
	CW_Valve_Not_Ready,
	Pump_Not_Ready
	
);
END_TYPE

// 80 Status Enums/Level_2/Temp_loop_Status
{attribute 'qualified_only'}
//{attribute 'strict'}
TYPE Temp_loop_Status :
(
	Idle:=0,
	Pre_Start,
	Crash,
	Ramping,
	Auto,
	Timed,
	Timer_Expired,
	Warning,
	HiHi_Alarm,
	HiHi_Warning,
	LoLo_Warning,
	LoLo_Alarm,
	OK,
	Paused,
	External_Fault,
	Valve_Not_auto,
	Sensor_Forced,
	Fault
);
END_TYPE

// 80 Status Enums/Level_2/Transfer_Status
{attribute 'qualified_only'}
//{attribute 'strict'}
{attribute 'to_string'}
TYPE Transfer_Status :
(
	IDLE := 0,
	Running,
	FIT_Reset,
	Open_Valve,
	Complete,
	VFD_Not_Ready,
	LOCKED_OUT,
	Paused,
	Valve_Not_Auto,
	Sensor_Forced,
	ACV_Not_Ready,
	BCV_Not_Ready,
	Flow_Meter_Active,
	Bypass,
	Pump_Not_Ready,
	Valve_Not_Ready,
	Flow_Active,
	Destination_Not_Ready,
	Disabled
);
END_TYPE

// 80 Status Enums/Level_3/eBatch_Status
{attribute 'qualified_only'}
{attribute 'to_string'}
TYPE eBatch_Status :
(
	Disabled := 0,
	PV_Not_Ready,
	CV_Not_Ready,
	Idle,
	Ready,
	FIT_Reset,
	Starting,
	Active,
	Ending,
	Complete,
	Paused,
	
	Fault
	
);
END_TYPE

// 80 Status Enums/Vessels/BH_Vessel_Status
{attribute 'qualified_only'}
//{attribute 'strict'}
TYPE BH_Vessel_Status :
(
	Off := 0,
	OK,
	Ramping,
	Controling,
	Timer_Active,
	Timer_Done,
	Zone_1_Error,
	Zone_2_Error,
	Zone_3_Error,
	Zone_4_Error,
	High_Alarm,
	High_Warning,
	Low_Warning,
	Low_Alarm
	
);
END_TYPE

// 80 Status Enums/Vessels/eBrite_Status
{attribute 'qualified_only'}
//{attribute 'strict'}
{attribute 'to_string'}
TYPE eBrite_Status :
(
	Sensor_Fault := 0,
	Valve_Fault,
	Coolant_Fault,
	IDLE,		//3
	On,			//4
	Regulating,
	Low_Warning,
	High_Warning,
	Low_Alarm,
	High_Alarm
);
END_TYPE

// 80 Status Enums/Vessels/eCLT_Status
{attribute 'qualified_only'}
//{attribute 'strict'}
{attribute 'to_string'}
TYPE eCLT_Status :
(
	OFF := 0,
	Active,
	Fault,
	Line_Chase_Reset_Flow_Meter,
	Line_Chase_Open_Valve,
	Line_Chase_Active,
	Line_Chase_Complete,
	Low_Tank_Level,
	High_Tank_Temperature,
	Cooling,
	OK,
	Low_Level,
	Low_Low_Level
);
END_TYPE

// 80 Status Enums/Vessels/eFermenter_Status
{attribute 'qualified_only'}
//{attribute 'strict'}
{attribute 'to_string'}
TYPE eFermenter_Status :
(
	Sensor_Fault := 0,
	Valve_Fault,
	Coolant_Fault,
	IDLE,		//3
	Regulating,		//4
	Crashing,		//5
	Low_Warning,
	High_Warning,
	Low_Alarm,
	High_Alarm
);
END_TYPE

// 80 Status Enums/Vessels/eGrain_Room_Status
{attribute 'qualified_only'}
//{attribute 'strict'}
{attribute 'to_string'}
TYPE eGrain_Room_Status :
(
	OFF := 0,
	Not_Ready,
	Wait_For_MM,
	Open_Hydrator,
	Start_Conveyor,
	Open_Hopper,
	Active,
	Complete,
	Close_Hopper,
	Stop_Conveyor,
	Close_Hyrdator,
	Scale_Not_Ready,
	Conveyor_Not_Ready,
	Hydrator_Not_Ready,
	Hopper_Not_Ready
	
);
END_TYPE

// 80 Status Enums/Vessels/eHLT_Status
{attribute 'qualified_only'}
//{attribute 'strict'}
{attribute 'to_string'}
TYPE eHLT_Status :
(
	OFF := 0,
	Active,
	Fault,
	Line_Chase_Reset_Flow_Meter,
	Line_Chase_Open_Valve,
	Line_Chase_Active,
	Line_Chase_Complete,
	Low_Tank_Level,
	Low_Tank_Temperature
);
END_TYPE

// 80 Status Enums/Vessels/eKT_Status
{attribute 'qualified_only'}
//{attribute 'strict'}
{attribute 'to_string'}
TYPE eKT_Status :
(
	IDLE := 0,
	System_Check,
	Ready,
	Start,
	Active,
	Complete,
	
	PreHeat,
	PreHeat_Complete,
	Opening_Wort_In_Valves,
	Start_Rocket,
	Rocket_Boil,
	Jacket_Boil,
	
	Full_Boil_Start,
	Full_Boil,
	Full_Boil_Complete,
	
	Waiting_For_Wort,
	Recieving_Wort,
	Enable_Rocket,
	Rocket_Active,
	Wort_Transfer_Start,
	Wort_Transfer_Active,
	Wort_Transfer_Complete,
	
	Transfer_Flush_Validate,
	Transfer_Flush_Active,				//
	Transfer_Flush_Complete,
	
	Holding_Temperature,
	Whirlpool_Start,
	WhirlPool_Active,
	Rest,
	Select_Fermenter,
	Enable_Cast_Out,
	CastOut,
	CastOut_Chase_Start,
	CastOut_Chase_Active,
	Rocket_Prepare,
	Rocket_Open_Vent,
	Rocket_Flood,
	Rocket_Drain,
	Drain_Complete,
	Tank_Rinse_Prepare,
	
	
	
	
	
	
	
	//////////////Alarms////////////////////
	
	KT_Chase_Valve_Not_Ready,
	KT_CIP_Recirc_Valve_Not_Ready,
	Pump_Chase_Valve_Not_Ready,
	KT_Pump_Drain_BCV_Valve_Not_Ready,
	KT_Rocket_Condensate_Valve_Not_Ready,
	KT_Rocket_Cooling_Isolation_Not_Ready,
	KT_Rocket_Cooling_Return_Valve_Not_Ready,
	KT_Rocket_Drain_Not_Ready,
	KT_Rocket_Shell_Drain_Not_Ready,
	KT_Rocket_Steam_Isolation_Not_Ready,
	KT_Spray_Ball_Chase_Valve_Not_Ready,
	KT_Tank_Bottom_Valve_Not_Ready,
	KT_TO_WP_Valve_Not_Ready,
	KT_Lower_Jacket_Steam_Valve_Not_Ready,
	KT_Middle_Jacket_Steam_Valve_Not_Ready,
	KT_Recirc_Valve_Not_Ready,
	KT_Rocket_Cooling_Control_Valve_Not_Ready,
	KT_Rocket_Steam_Control_Valve_Not_Ready,
	KT_Upper_Jacket_Steam_Valve_Not_Ready,
	KT_Lower_Jacket_PID_Not_Ready,
	KT_Middle_Jacket_PID_Not_Ready,
	KT_Rocket_Cooling_PID_Not_Ready,
	KT_Rocket_Heating_PID_Not_Ready,
	KT_Upper_Jacket_PID_Not_Ready,
	KT_Discharge_Temperature_Not_Ready,
	KT_Rocket_Discharge_Temperature_Not_Ready,
	KT_Vesel_Temperature_Not_Ready,
	//KT_Agitator_Not_Ready,
	//KT_Discharge_Pump_Not_Ready,
	KT_Condensate_Return_Valve_Not_Ready,
	KT_Rocket_Condensate_Return_Valve_Not_Ready,
	//Waiting_For_Wort,
	Enable_Lower_Jacket,
	Enable_Middle_Jacket,
	Enable_Upper_Jacket,
	//Enable_Rocket,
	Rocket_Empty,
	Rocket_No_Flow,
	Discharge_Pump_Not_Ready,
	Agitator_Not_Ready,
	Discharge_Pump_Intake_Empty,
	Rocket_Condensate_Fault,
	Jacket_Condensate_Fault,
	Whirlpool_Not_In_Auto,
	Whirlpool_Not_Idle,
	Drain_Active,
	Wort_In_Enable_Rocket,
	Wort_In_Rocket,
	Rinse,
	Rinse_Complete,
	Rinse_Tangent,
	Rinse_High_Outlet,
	Rinse_Low_Outlet,
	Rinse_Tank,
	Drain_1,
	Drain_2,
	Drain_3
	
	
	
);
END_TYPE

// 80 Status Enums/Vessels/eLT_Status
{attribute 'qualified_only'}
//{attribute 'strict'}
{attribute 'to_string'}
TYPE eLT_Status :
(
	IDLE := 0,
	Recipe_Copied,
	LauterTun_Check,
	LauterTun_Ready,
	Foundation_Water_Prepare,						//
	Foundation_Water,			//
	Foundation_Water_Complete,
	Mash_In_Check,
	Mash_In_Ready,	//
	Mash_In_Active,					//
	Mash_In_Complete,
	
	Underlet_Validate,
	UnderLet_Ready,			//
	Underlet_Active,					//
	Underlet_Complete,			//
	Underlet_Resting,						//
	Underlet_Rest_Complete,
	Underlet_Agitate,

	Vorlauf_Validate,
	Vorlauf_Ready,
	Raise_Plough,
	Vorlauf_Active,				//
	Vorlauf_Complete,
	
	Transfer_Validate,
	Transfer_Ready,
	Clear_FloWave_Volume,
	Transfer_Active,
	Transfer_Complete,
		
	Transfer_Sparge_Validate,
	Transfer_Sparge_Ready,
	Transfer_Sparge_Start,					//
	Transfer_Sparge_Active,
	Sparge_Complete_Waiting_on_Transfer,
	Transfer_Complete_Waiting_on_Sparge,
	Transfer_Sparge_Complete,			//
	
	Transfer_Empty_Validate,
	Transfer_Empty_Ready,
	Transfer_Empty_Running,
	Transfer_Min_Time_Complete,
	Transfer_Empty_Complete,
		//			//
	Transfer_Flush_Validate,
	Transfer_Flush_Active,				//
	Transfer_Flush_Complete,
	
	Tank_Clean_Active,
	Tank_Clean_Complete,
	
	Rinse_Active,				//
	Rinse_Complete,
			//
	Drain,						//
	Drain_Complete,
	
	Grain_out_Active,
	Raise_Elevator,
	Lower_Plough,
	Open_Grain_Door,
	Active,
	Complete,
	CIP_Active,
	Systems_Check,


	Validate,
	Ready,
	Resting,

	Open_KT_Supply_Valve,
	Low_Air,
	Low_Steam,
	Low_Pressure,
	Low_Flow,
	Rake_Not_Ready,
	Rake_Adjust_Not_Ready,
	Plough_Not_Ready,
	Pump_Not_Ready,
	Valves_Not_In_Auto,
	Jacket_Not_In_Auto,
	Sparge_Not_Ready,
	Grain_Door_Not_Closed,
	MT_To_LT_Valve_Not_In_Auto,
	Underlet_Not_Available,
	Grant_Supply_Control_Not_Ready,
	Grant_Discharge_Control_Not_Ready,
	Sparge_Transfer_Not_Ready,
	Grant_Supply_Valve_Not_Ready,
	Grant_Discharge_Valve_Not_Ready,
	Grant_Level_Sensor_Error,
	LT_to_KT_Transfer_Not_Ready,
	Sparge_Mix_Not_Ready,
	Flush_Not_Ready,
	Paused,
	Kettle_Not_In_Auto,
	Kettle_Not_Idle,
	
	PreHeat_Active,
	PreHeat_Complete,
	
	Vorlauf_Low_Flow,
	Grain_Out_Complete,
	
	Rinse_Tank,
	Rinse_Sprayball_A,
	Rinse_Sprayball_A_B,
	Rinse_Sprayball_B,
	Rinse_Sprayball_B_A,
	Rinse_Tank_Complete,
	Rinse_Grant,
	Rinse_Grant_Active,
	Rinse_Grant_Complete,
	Close_Grain_Door,
	Rinse_Underlet,
	Rinse_Underlet_Active
	

		
);
END_TYPE

// 80 Status Enums/Vessels/eMM_Status
{attribute 'qualified_only'}
//{attribute 'strict'}
{attribute 'to_string'}
TYPE eMM_Status :
(
	IDLE := 0,
	Waiting_For_Brew_Confirmation,
	PreHeat_Validate,
	PreHeat_Ready,
	PreHeating_Vessel,
	PreHeat_Complete,
	Mash_In_Validate,
	Mash_In_Ready,
	Foundation_Water,
	Grain_Dispense,
	Grain_Rinse,
	Mash_In_Complete,
	Heat_Profile_1_Active,
	Heat_Profile_1_Complete,
	Heat_Profile_2_Active,
	Heat_Profile_2_Complete,
	Heat_Profile_3_Active,
	Heat_Profile_3_Complete,
	Heat_Profile_4_Active,
	Mash_Out_Validate,
	Mash_Out_Ready,
	Waiting_to_Transfer,
	Open_Transfer_Valve,
	Transfer_1,
	Transfer_Rest_1,
	Transfer_2,
	Transfer_Rest_2,
	Transfer_3,
	Transfer_Complete,
	Transfer_Chase_Validate,
	Transfer_Chase_Ready,
	Transfer_Chase_Active,
	Transfer_Chase_Complete,
	Mash_Out_Complete,
	Tank_Rinse_Validate,
	Tank_Rinse_Ready,
	Tank_Rinse_Active,
	Tank_Rinse_Complete,
	Tank_Drain,
	Tank_Drain_Complete,
	
	
	
	
	
	
	Low_Steam,
	Low_Air,
	Upper_Jacket_Not_In_Auto,
	Middle_Jacket_Not_In_Auto,
	Lower_Jacket_Not_In_Auto,
	Upper_Jacket_Valve_Not_In_Auto,
	Middle_Jacket_Valve_Not_In_Auto,
	Lower_Jacket_Valve_Not_In_Auto,
	Grain_Hopper_Valve_Not_In_Auto,
	Strike_Water_System_Not_Ready,
	
	LT_Not_In_Auto,
	LT_Grain_Door_Not_Closed,
	LT_Agitator_Not_Ready,
	LT_Rake_Not_Ready,
	LT_Pump_Not_Ready,
	LT_Sparge_Not_Ready,
	Line_Chase_Not_Available,
	LT_Not_Waiting_For_Mash,
	Rinse_Valve_A,
	Rinse_Valve_A_B,
	Rinse_Valve_B,
	Rinse_Valve_B_A,
	
	//Extra's added to accomadate MLT
	Vorlauf_Active,
	Vorlauf_Complete,
	Sparge_Active,
	Sparge_Complete,
	Underlet_Start,
	Underlet_Active,
	Underlet_Complete,
	Grain_Out,
	Grain_Out_Complete,
	Rinse_Grant,
	Rinse_Underlet,
	Rinse_Vessel,
	Underlet_Mix,
	Underlet_Rest,
	
	

	MM_Status_End
);
END_TYPE

// 80 Status Enums/Vessels/eWP_Status
{attribute 'qualified_only'}
//{attribute 'strict'}
{attribute 'to_string'}
TYPE eWP_Status :
(
	IDLE := 0,
	Recipe_Copy,
	Ready_For_Wort,
	Whirpool_Validate,
	WhirlPool_Active,
	Whirpool_Complete,
	Ready,
	Running,
	Active,
	Profile_2,
	Profile_3,
	Cast_out_1,
	Profile_4,
	Resting,
	Rest_Complete,
	Select_Fermenter,
	Fermenter_Capacity_Error,
	CastOut_Validate,
	CastOut_Start,
	CastOut_Active,
	CastOut_Complete,
	Chase_Validate,
	Chase_Active,
	Chase_Complete,
	Rinse_Validate,
	Rinse_Active,
	Rinse_Complete,

	Pump_Not_Ready,
	Trub_Rinse_Validate,
	Trub_Rinse_active,
	Trub_Rinse_Drain,
	Trub_Rinse_Complete,
	Drain_Active,
	Drain_Complete
	
	
	
	
);
END_TYPE

// 90 Task Enums/Level_3/eBatch_Task
{attribute 'qualified_only'}
//{attribute 'strict'}
{attribute 'to_string'}
TYPE eBatch_Task :
(
	OFF := 0,
	Run,
	Pause,
	Resume
	
);
END_TYPE

// 20 Program Organization Units/Level_0_Remote_IO/CanOpen/cSDO_DUT
TYPE cSDO_DUT :
STRUCT
	NodeId:BYTE;
	Index:WORD;
	SubIndex:BYTE;
	Bytes:WORD;
	Data:ARRAY[0..3] OF BYTE;
	Read:BOOL;
	Write:BOOL;
	Done:BOOL;
	Busy:BOOL;
	Error:BOOL;
	
	
END_STRUCT
END_TYPE

// 30 Visualizations/VISU
{attribute 'qualified_only'}
VAR_GLOBAL
	Vessel_Index:INT:=0;
	Total_Vessels:INT:=10;
	Tank_Farm_Y_Offset:INT:=150;
	Tank_Farm_X_Offest:INT:=300;
	Tank_Farm_width:INT:=1024;
	Tank_Farm_Height:INT:=768;
	Tank_Farm_X_Count:INT:=3;
	Tank_Farm_y_Count:INT:=5;
	Tank_Farm_Positions:ARRAY[0..100] OF ARRAY[0..3] OF INT;
END_VAR

// 40 Data Types/Base_Declarations/ASI
{attribute 'qualified_only'}
VAR_GLOBAL
	CH1_Flags:ARRAY[0..7] OF DWORD;
	CH1_Analog_1_RX:ARRAY[0..79] OF WORD;
	CH1_Analog_2_RX:ARRAY[0..74] OF WORD;
	CH1_Analog_1_TX:ARRAY[0..79] OF WORD;
	CH1_Analog_2_TX:ARRAY[0..74] OF WORD;
	CH1_Digital_RX:ARRAY[0..63] OF BYTE;
	CH1_Digital_TX:ARRAY[0..63] OF BYTE;
	
	Master_1_Ch1_A:ARRAY[1..32] OF Asi_Node_DUT;
	Master_1_Ch1_B:ARRAY[1..32] OF Asi_Node_DUT;


	CH2_Flags:ARRAY[0..7] OF DWORD;
	CH2_Analog_1_RX:ARRAY[0..79] OF WORD;
	CH2_Analog_2_RX:ARRAY[0..74] OF WORD;
	CH2_Analog_1_TX:ARRAY[0..79] OF WORD;
	CH2_Analog_2_TX:ARRAY[0..74] OF WORD;
	CH2_Digital_RX:ARRAY[0..63] OF BYTE;
	CH2_Digital_TX:ARRAY[0..63] OF BYTE;
	
	Master_1_Ch2_A:ARRAY[1..32] OF Asi_Node_DUT;
	Master_1_Ch2_B:ARRAY[1..32] OF Asi_Node_DUT;
	
	AC2916:ARRAY[0..AC2916_Mapping.AC2916_End] OF AC2916_DUT;
END_VAR

// 40 Data Types/Base_Declarations/GVL
{attribute 'qualified_only'}
VAR_GLOBAL
	(*
	HMI_Cellar_Index:INT:=255;
	HMI_Cellar_Data:cFermenter_DUT;
	
	
	HMI_Brite_Index:INT:=155;
	HMI_Brite_Data:cBrite_DUT;
	
	HMI_TT_Index:INT:=255;
	HMI_TT_Data:AIT_DUT;
	
	HMI_AIT_Index:INT:=255;
	HMI_AIT_Data:AIT_DUT;
	
	HMI_PT_Index:INT:=255;
	HMI_PT_Data:AIT_DUT;
	
	HMI_FIT_Index:INT:=255;
	HMI_FIT_Data:FIT_DUT;
	
	HMI_PID_Index:INT:=255;
	HMI_PID_Data:PID_DUT;
	
	
	HMI_ACV_Index:INT:=255;
	HMI_ACV_Data:ACV_DUT;
	ACV:ARRAY[0..ACV_Mapping.ACV_End] OF ACV_DUT;
	
	
	HMI_VFD_INDEX:INT;
	HMI_VFD_DATA:VFD_Vacon_DUT;
	Vacon_VFD:ARRAY[0..Vacon_VFD_Mapping.Vacon_End] OF VFD_Vacon_DUT;
	
	
	
	HMI_BCV_Index:INT:=255;
	HMI_BCV_Data:BCV_DUT;
	BCV:ARRAY[0..BCV_Mapping.BCV_End] OF BCV_DUT;
	
	
	HMI_LS_Index:INT:=255;
	HMI_LS_Data:DI_DUT;
	LS:ARRAY[0..LS_Mapping.LS_END] OF DI_DUT;
	
	HMI_Condensate_Index:INT;
	HMI_Condensate_Data:cCondensate_Trap;
	
	HMI_Index_Reset:BOOL;
	
	RTC : SysTimeDate;
	
	Day_Seconds:UDINT;
	
	//HMI_Transfer_Index:INT;
	//HMI_Transfer_Data:cChase;
	
	
	HMI_qMix_Index:INT:=255;
	HMI_qMix_Data:Quick_Mix_Dut;
	
	Transfer_Active:BOOL;
	//MLT_Mode:INT;
	//MLT_Task:INT;
	//HMI_Ticker:WORD;
	
	//BaseTopic:STRING:='cornel/';
	Dout:ARRAY[0..Dout_mapping.Do_End] OF DO_DUT;
	*)
	
END_VAR

// 40 Data Types/Base_Declarations/HMI
{attribute 'qualified_only'}
VAR_GLOBAL
	Ref_cAlarm:REFERENCE TO cAlarm_Config;
	
	HMI_8050_Index:INT:=255;
	HMI_8050_data:REFERENCE TO HMI_8050;
	
END_VAR

// 40 Data Types/Base_Declarations/Network
{attribute 'qualified_only'}
VAR_GLOBAL
	MLT_agitator:Vacon_MbTCP;
	MLT_Pump:Vacon_MbTCP;
	HLT_Mix:Vacon_MbTCP;
	HLT_Recirc:Vacon_MbTCP;
	KTWP_Discharge:Vacon_MbTCP;
	
	

END_VAR

// 40 Data Types/Base_Declarations/PVL
{attribute 'qualified_only'}
VAR_GLOBAL
	//Fermenter:ARRAY[0..1] OF cFermenter_DUT;
	//Brite:ARRAY[0..Brite_mapping.Brite_End] OF cBrite_DUT;
	
	//Config:Config_DUT;
	//qMix:ARRAY[0..Mix_Mapping.Mix_End] OF Quick_Mix_DUT;
//	TT:ARRAY[0..TT_Mapping.TT_End] OF AIT_DUT;
//	AIT:ARRAY[0..AIT_Mapping.AIT_End] OF  AIT_DUT;
	//PT:ARRAY[0..PT_Mapping.PT_End] OF  AIT_DUT;
	//FIT:ARRAY[0..FIT_Mapping.FIT_END] OF FIT_DUT;
	//PID:ARRAY[0..PID_Mapping.PID_END] OF PID_DUT;
	//Mix:ARRAY[0..Mix_Mapping.Mix_End] OF Mix_DUT;
END_VAR

// 40 Data Types/Base_Declarations/RIO
{attribute 'qualified_only'}
VAR_GLOBAL
	//Di:ARRAY[0..3] OF BYTE;
	Di:ARRAY[0..4] OF BYTE;
	
	Dout:ARRAY[0..1] OF BYTE;
	AI:ARRAY[0..5] OF ARRAY[0..3] OF WORD;
	HSC_In:ARRAY[0..2] OF ARRAY[0..3] OF WORD;
	HSC_Out:ARRAY[0..2]OF ARRAY[0..3] OF WORD;
	
END_VAR

// 20 Program Organization Units/ACV_Temp_Loop_UDFB
FUNCTION_BLOCK ACV_Temp_Loop_UDFB
VAR_IN_OUT
	ACV_LOOP: ACV_Temp_Loop_DUT;
	ACV:ACV_DUT;
	TT:AIT_DUT;

END_VAR

VAR_INPUT
	Heating: BOOL;
	LOCKOUT:BOOL:=FALSE;
	Permisive:BOOL:=TRUE;
	External_Fault:BOOL:=FALSE;
END_VAR
VAR

	FT_PID_0: BURKERT_OSCAT_BASIC.CTRL_PID;
	GEN_PULSE_0: BURKERT_OSCAT_BASIC.GEN_PULSE;
	In_Zone: BOOL;
	TON_0: TON;
	R_TRIG_0: R_trig;
	Timer_Status: INT;
	ABS_Error: REAL;
	R_TRIG_1: R_trig;
	RAMP_REAL_0: Util.RAMP_REAL;
	SR_0: SR;
	TON_1: TON;
	TOF_0: TOF;
	TON_2: TON;
	FT_PID_1:Util.PID_FIXCYCLE;
	Temp_Loop_PID:BOOL:=TRUE;
	R_trig_2:R_Trig;
	Loop_Disable:BOOL;
	TP_1:TP;
	
	FT_PIDW_1: BURKERT_OSCAT_BASIC.FT_PIDW;
END_VAR
VAR_OUTPUT

END_VAR
VAR // added by the converter: edge detectors and wires of the graphical bodies
    _w1, _w2, _w3, _w4, _w5, _w6, _w7, _w8, _w9, _w10, _w11, _w12, _w14 : ANY;
    _w13 : TIME;
END_VAR

// note: 7 stored wires end on pins the file does not list and are not shown
ACV_Loop.DeadBand := SEL(ACV_Loop.DeadBand = 0.0, ACV_Loop.DeadBand, 0.1);
ACV_Loop.Live_Target_EU := SEL(ACV_Loop.Mode=Temp_Loop_Modes.Step, ACV_Loop.Target_EU, SEL(HEATING, TT.EU-(ACV_Loop.DeadBand*1.5), TT.EU+(ACV_Loop.DeadBand*1.5)));
_w1 := (ACV_Loop.Mode = Temp_Loop_Modes.Crash) OR (ACV_Loop.Mode = Temp_Loop_Modes.Step);
_w2 := ABS(ACV_Loop.Target_Eu - TT.EU);
ABS_Error := _w2;
(* _w2 * ACV_Loop.kp < 50; result not used *)
TON_2(IN := False OR _w2 < (ACV_Loop.DeadBand*4), PT := T#5s); // TON
_w3 := _w1 AND TON_2.Q;
In_Zone := _w3;
R_TRIG_0(CLK := _w1 AND _w3); // R_trig
IF R_TRIG_0.Q THEN _w4 := Temp_Loop_Modes.Auto; END_IF
ACV_Loop.Mode := _w4;
_w5 := SEL(Heating, ACV_Loop.Live_Target_EU, ACV_Loop.Actual_EU);
ACV_Loop.Int_Out := FT_PIDW_1.YI;
_w6 := SEL(Heating, ACV_Loop.Actual_EU, ACV_Loop.Live_Target_EU);
TOF_0(IN := Permisive, PT := T#5s); // TOF
SR_0(SET1 := Loop_Disable, RESET := ACV_Loop.Mode=Temp_Loop_Modes.Idle); // SR
_w7 := (ACV_Loop.Mode=Temp_Loop_Modes.Auto_Paused) OR (ACV_Loop.Mode=Temp_Loop_Modes.Idle) OR NOT TOF_0.Q OR SR_0.Q1 OR (ACV_Loop.Status=Temp_Loop_Status.Timer_Expired) OR (TT.Status.eStatus=eSensor_Status.Offline) OR (TT.Status.eStatus=eSensor_Status.Fault) OR (acv.Status=eACV_Status.OFFLINE);
_w8 := SEL(_w7, _w6, _w5) - _w5;
TP_1(IN := _w3, PT := T#5s); // TP
FT_PIDW_1(
    IN := _w8,
    KP := ACV_Loop.kp,
    TN := ACV_Loop.TN,
    TV := ACV_Loop.TV,
    LIM_L := 0,
    LIM_H := 100,
    RST := _w7 OR TP_1.Q); // BURKERT_OSCAT_BASIC.FT_PIDW
ACV_Loop.Limiter := FT_PIDW_1.LIM;
_w9 := SEL(ACV_Loop.Mode=Temp_Loop_Modes.Crash, FT_PIDW_1.Y, 100.0);
ACV_Loop.Diff_Out := FT_PIDW_1.diff.out;
_w10 := SEL(Loop_Disable, _w9, 0.0);
ACV.PLC_CMD := _w10;
ACV_Loop.Load_EU := _w10;
IF SR_0.Q1 THEN _w11 := Temp_Loop_Modes.Idle; END_IF
ACV_Loop.Mode := _w11;
TT.Alarm_Config.Setpoints.Hi_Hi_Alarm := SEL(NOT _w7, TT.Alarm_Config.Setpoints.Hi_Hi_Alarm, ACV_Loop.Live_Target_EU+(ACV_Loop.Window*2));
TT.Alarm_Config.Setpoints.Hi_Warn := SEL(NOT _w7, TT.Alarm_Config.Setpoints.Hi_Warn, ACV_Loop.Live_Target_EU+(ACV_Loop.Window));
TT.Alarm_Config.Setpoints.Low_warn := SEL(NOT _w7, TT.Alarm_Config.Setpoints.Low_warn, ACV_Loop.Live_Target_EU-(ACV_Loop.Window));
TT.Alarm_Config.Setpoints.Low_Low_Alarm := SEL(NOT _w7, TT.Alarm_Config.Setpoints.Low_Low_Alarm, ACV_Loop.Live_Target_EU-(ACV_Loop.Window*2));
ACV_Loop.Actual_EU := TT.EU;
ACV_Loop.Error_EU := SEL(ACV_Loop.Mode=Temp_Loop_Modes.Idle, TT.EU - ACV_Loop.Target_EU, 0.0);
_w12 := (ACV_Loop.Mode=Temp_Loop_Modes.Auto) AND (ACV_Loop.Timer_Target_M>0);
_w13 := UINT_TO_TIME(ACV_Loop.Timer_Target_M) * 60000;
TON_0(IN := _w12, PT := _w13); // TON
ACV_Loop.Timer_Remaining_s := TIME_TO_UINT((_w13 - TON_0.ET) / 1000);
_w14 := (TT.Status.eStatus=eSensor_Status.Offline) OR (TT.Status.eStatus=eSensor_Status.Fault) OR (acv.Status=eACV_Status.OFFLINE);
Loop_Disable := External_Fault OR (TT.Status.eStatus=eSensor_Status.FORCED) OR (ACV.Mode<>ACV_Modes.Auto) OR _w14;
ACV_Loop.Status := SEL(ACV.Mode<>ACV_Modes.Auto, SEL(TT.Status.eStatus=eSensor_Status.FORCED, SEL(External_Fault, SEL(_w14, SEL(ACV_Loop.Mode=Temp_Loop_Modes.Auto_Paused, SEL(ACV_Loop.Mode=Temp_Loop_Modes.Idle, SEL(TT.Status.eStatus=eSensor_Status.Low_Low_Alarm, SEL(TT.Status.eStatus=eSensor_Status.Low_Warning, SEL(TT.Status.eStatus=eSensor_Status.HiHi_Alarm, SEL(TT.Status.eStatus=eSensor_Status.High_Warning, SEL(TON_0.Q, SEL(_w12, SEL(ACV_Loop.Mode=Temp_Loop_Modes.Auto, SEL(Permisive, Temp_Loop_Status.Pre_Start, Temp_Loop_Status.Ramping), Temp_Loop_Status.Auto), Temp_Loop_Status.Timed), Temp_Loop_Status.Timer_Expired), Temp_Loop_Status.HiHi_Warning), Temp_Loop_Status.HiHi_Alarm), Temp_Loop_Status.LoLo_Warning), Temp_Loop_Status.LoLo_Alarm), Temp_Loop_Status.Idle), Temp_Loop_Status.Paused), Temp_Loop_Status.Fault), Temp_Loop_Status.External_Fault), Temp_Loop_Status.Sensor_Forced), Temp_Loop_Status.Valve_Not_auto);
// TRUE: input not connected
// Temp_Loop_Status.Idle: input not connected

END_FUNCTION_BLOCK

// 20 Program Organization Units/Basic_Temp_LOOP
FUNCTION_BLOCK Basic_Temp_LOOP
VAR	
	RS_0: RS;
END_VAR
VAR_IN_OUT
	Loop:BCV_Temp_Loop_DUT;
END_VAR
VAR_INPUT
END_VAR
VAR // added by the converter: edge detectors and wires of the graphical bodies
    _w1 : ANY;
END_VAR

_w1 := Loop.Target_EU + Loop.Window;
RS_0(SET := loop.Actual_EU > Loop.DeadBand + _w1, RESET1 := loop.Actual_EU < _w1 - Loop.DeadBand); // RS
Loop.Output := RS_0.Q1;

END_FUNCTION_BLOCK

// 20 Program Organization Units/BCV_Temp_Loop_UDFB
FUNCTION_BLOCK BCV_Temp_Loop_UDFB
VAR_IN_OUT
	BCV_LOOP: BCV_Temp_Loop_DUT;
	BCV:BCV_DUT;
	TT:AIT_DUT;

END_VAR

VAR_INPUT
	Heating: BOOL;
	LOCKOUT:BOOL:=FALSE;
	Permisive:BOOL:=TRUE;
	External_Fault:BOOL:=FALSE;
	//Temp_Loop_PID:WORD:=2;
	//BCV_ID:INT;
	//TT_ID:INT;
END_VAR
VAR

	FT_PID_0: BURKERT_OSCAT_BASIC.CTRL_PID;
	GEN_PULSE_0: BURKERT_OSCAT_BASIC.GEN_PULSE;
	In_Zone: BOOL;
	TON_0: TON;
	R_TRIG_0: R_trig;
	Timer_Status: INT;
	ABS_Error: REAL;
	R_TRIG_1: R_trig;
	RAMP_REAL_0: Util.RAMP_REAL;
	SR_0: SR;
	TON_1: TON;
	TOF_0: TOF;
	TON_2: TON;
	FT_PID_1:Util.PID_FIXCYCLE;
	
	R_trig_2:R_Trig;
	Loop_Disable:BOOL;
	TP_1:TP;
	
	FT_PIDWL_0: BURKERT_OSCAT_BASIC.FT_PIDWL;
	FT_PIDW_0: BURKERT_OSCAT_BASIC.FT_PIDW;
	TOF_1: TOF;
	On_Seconds: REAL;
	PID_Reset: BOOL;
	TON_3: TON;
	TP_0: TP;
	Current_Minute: UINT;
	R_TRIG_3: R_trig;
	TON_4: TON;
	Profile_Reset: BOOL;
END_VAR
VAR_OUTPUT

END_VAR
VAR // added by the converter: edge detectors and wires of the graphical bodies
    _w1, _w2, _w3, _w4, _w7, _w8, _w10, _w12, _w13, _w14, _w15, _w19, _w21, _w23, _w25, _w27 : ANY;
    _w5, _w11 : TIME;
    _w6, _w9, _w16, _w17, _w18, _w20, _w22, _w24, _w26 : BOOL;
END_VAR

